(* CODESYS project mobject-core.library
   Author: mobject dev team
   Version: 0.10.0
   Title: mobject-core
   Placeholder: mobject-core
   DefaultNamespace: mobject-core
   Company: mobject

Project tree, tasks and I/O mapping:
  libraries: Tc2_Standard, * (Beckhoff Automation GmbH); Tc2_System, * (Beckhoff Automation GmbH); Tc2_Utilities, * (Beckhoff Automation GmbH); Tc3_JsonXml, * (Beckhoff Automation GmbH)
  mobject-collections/
    _Internal/
      Dictionary/
        Enumerator/
          function block DictionaryForwardEnumerator [ST]: FB_init, FB_exit, HandleEvent, IsValid, Key, MoveNext, Reset, TryGet, TryGetTo
        Node/
          function block DictionaryTreeNode [ST]: FB_init, FB_exit, CopyBufferToDestination, CopySourceToBuffer, CreateBuffer, DestroyBuffer, DataSize, DeepCopy, Equals, Height, Key, Left, NodeBufferPointer, NodeBufferSize, Reinitialize, Right, TryGet, TryGetTo
      Events/
        Collection/
          function block CollectionChangedEvent [ST]
          function block CollectionDisposedEvent [ST]
          function block CollectionEvent [ST]: FB_init, Target
        KeyValueCollection/
          function block KeyValueCollectionChangedEvent [ST]
          function block KeyValueCollectionDisposedEvent [ST]
          function block KeyValueCollectionEvent [ST]: FB_init, Target
      LinkedList/
        Enumerator/
          function block LinkedListForwardEnumerator [ST]: FB_init, FB_exit, HandleEvent, IsValid, MoveNext, Reset, TryGet, TryGetTo
        Node/
          function block LinkedListNode [ST]: FB_init, FB_exit, CopyBufferToDestination, CopySourceToBuffer, CreateBuffer, DestroyBuffer, DataSize, Equals, Next, Previous, TryGet, TryGetTo
      OrderedDictionary/
        Enumerator/
          function block OrderedDictionaryForwardEnumerator [ST]: FB_init, FB_exit, HandleEvent, IsValid, Key, MoveNext, Reset, TryGet, TryGetTo
        Node/
          function block OrderedDictionaryTreeNode [ST]: FB_init, FB_exit, CopyBufferToDestination, CopySourceToBuffer, CreateBuffer, DestroyBuffer, DataSize, DeepCopy, Equals, Height, Key, Left, Next, NodeBufferPointer, NodeBufferSize, Previous, Reinitialize, Right, TryGet, TryGetTo
      PriorityQueue/
    Dictionary/
      function block Dictionary [ST]: FB_exit, Balance, EmitChangedEvent, EmitDisposedEvent, FindMinimum, GetBalanceFactor, GetHeight, LeftRotate, RecursiveAddKeysInOrderToCollection, RecursiveAddNodesInOrderToCollection, RecursiveClear, RecursiveCountNodes, RecursiveDelete, RecursiveFind, RecursiveInsert, RightRotate, UpdateHeight, AddOrUpdate, Clear, ContainsKey, Count, GetEnumerator, GetKeys, GetKeyValueEnumerator, IsEmpty, OffEvent, OnceEvent, OnEvent, Remove, TryAdd, TryGetValue, TryGetValueTo
    Interfaces/
      Collections/
        Events/
          interface I_CollectionChangedEvent: Target
          interface I_CollectionDisposedEvent: Target
        Nodes/
          interface I_CollectionNode: DataSize, Equals, TryGet, TryGetTo
          interface I_LinkedListNode: Next, Previous
          interface I_ListNode
        interface I_Collection: AddItem, Clear, Contains, Count, IsEmpty, TryCopyTo, TryCopyToLocation, TryRemoveItem
        interface I_LinkedList: AddAfter, AddBefore, AddFirst, AddLast, Find, FindLast, First, Last, Remove, RemoveFirst, RemoveLast
        interface I_List: Capacity, GetIndexOf, TrimExcess, TryGetByIndex, TryGetToByIndex, TryInsert, TryRemoveAt
        interface I_Queue: Enqueue, TryDequeue, TryPeek
        interface I_Stack: Push, TryPeek, TryPop
      KeyValueCollections/
        Events/
          interface I_KeyValueCollectionChangedEvent: Target
          interface I_KeyValueCollectionDisposedEvent: Target
        Nodes/
          interface I_DictionaryTreeNode: DeepCopy, Height, Key, Left, NodeBufferPointer, NodeBufferSize, Reinitialize, Right
          interface I_OrderedDictionaryTreeNode: DeepCopy, Height, Key, Left, Next, NodeBufferPointer, NodeBufferSize, Previous, Reinitialize, Right
        interface I_Dictionary: AddOrUpdate, Clear, ContainsKey, GetKeys, IsEmpty, Remove, TryAdd, TryGetValue, TryGetValueTo
        interface I_KeyValueCollection
    LinkedList/
      function block LinkedList [ST]: FB_exit, AddNodeAfter, AddNodeBefore, AddNodeFirst, AddNodeLast, ContainsLinkedListNode, CreateNode, EmitChangedEvent, EmitDisposedEvent, FindFirstNodeWithValue, FindLastNodeWithValue, RemoveAllNodes, RemoveNode, AddAfter, AddBefore, AddFirst, AddItem, AddLast, Clear, Contains, Count, Find, FindLast, First, GetEnumerator, IsEmpty, Last, OffEvent, OnceEvent, OnEvent, Remove, RemoveFirst, RemoveLast, TryCopyTo, TryCopyToLocation, TryRemoveItem
    OrderedDictionary/
      function block OrderedDictionary [ST]: FB_exit, AddKeysInOrderToCollection, AddNodesInOrderToCollection, AddNodeToEnd, Balance, EmitChangedEvent, EmitDisposedEvent, FindMinimum, GetBalanceFactor, GetHeight, LeftRotate, RecursiveCountNodes, RecursiveDelete, RecursiveFind, RecursiveInsert, RemoveNodeFromLinkedList, ReplaceNodeInLinkedList, RightRotate, UpdateHeight, AddOrUpdate, Clear, ContainsKey, Count, GetEnumerator, GetKeys, GetKeyValueEnumerator, IsEmpty, OffEvent, OnceEvent, OnEvent, Remove, TryAdd, TryGetValue, TryGetValueTo
    Queue/
      function block Queue [ST]: FB_exit, EmitChangedEvent, EmitDisposedEvent, AddItem, Clear, Contains, Count, Enqueue, GetEnumerator, IsEmpty, OffEvent, OnceEvent, OnEvent, TryCopyTo, TryCopyToLocation, TryDequeue, TryPeek, TryRemoveItem
    Stack/
      function block Stack [ST]: FB_exit, EmitChangedEvent, EmitDisposedEvent, AddItem, Clear, Contains, Count, GetEnumerator, IsEmpty, OffEvent, OnceEvent, OnEvent, Push, TryCopyTo, TryCopyToLocation, TryPeek, TryPop, TryRemoveItem
  mobject-commands/
    _Internal/
      AsyncCommandStateMachine/
        function block AsyncCommandStateMachine [ST]: StateComplete_Aborting, StateComplete_Completing, StateComplete_Executing, StateComplete_Initializing, Abort, Error, ErrorId, Execute, IsAborted, IsAborting, IsCompleted, IsCompleting, IsErrored, IsExecuting, IsIdle, IsInitializing, Next
        interface I_AsyncCommandStateControl: Error, Next
    AsyncCommand/
      Interface/
        interface I_AsyncCommand: Abort, Busy, CyclicCall, Done, Error, ErrorId
      Runners/
        function block SingleAsyncCommandRunner [ST]: Busy, CyclicCall, Done, Error, ErrorId, ExecuteCommand
      function block AsyncCommand [ST]: OnAborted, OnAborting, OnCompleted, OnCompleting, OnErrored, OnExecuting, OnIdle, OnInitializing, Abort, Busy, CyclicCall, Done, Error, ErrorId, Execute
    Command/
      Interface/
        interface I_Command: Execute
  mobject-constants/
    global variables DatatypeLimits
  mobject-converters/
    Converters/
      BOOL_TO_/
        function TryConvert_BOOL_TO_BOOL [ST]
        function TryConvert_BOOL_TO_BYTE [ST]
        function TryConvert_BOOL_TO_DATE [ST]
        function TryConvert_BOOL_TO_Destination [ST]
        function TryConvert_BOOL_TO_DINT [ST]
        function TryConvert_BOOL_TO_DT [ST]
        function TryConvert_BOOL_TO_DWORD [ST]
        function TryConvert_BOOL_TO_INT [ST]
        function TryConvert_BOOL_TO_LINT [ST]
        function TryConvert_BOOL_TO_LREAL [ST]
        function TryConvert_BOOL_TO_LWORD [ST]
        function TryConvert_BOOL_TO_REAL [ST]
        function TryConvert_BOOL_TO_SINT [ST]
        function TryConvert_BOOL_TO_STRING [ST]
        function TryConvert_BOOL_TO_TIME [ST]
        function TryConvert_BOOL_TO_TOD [ST]
        function TryConvert_BOOL_TO_UDINT [ST]
        function TryConvert_BOOL_TO_UINT [ST]
        function TryConvert_BOOL_TO_ULINT [ST]
        function TryConvert_BOOL_TO_USINT [ST]
        function TryConvert_BOOL_TO_WORD [ST]
      BYTE_TO_/
        function TryConvert_BYTE_TO_BOOL [ST]
        function TryConvert_BYTE_TO_BYTE [ST]
        function TryConvert_BYTE_TO_DATE [ST]
        function TryConvert_BYTE_TO_Destination [ST]
        function TryConvert_BYTE_TO_DINT [ST]
        function TryConvert_BYTE_TO_DT [ST]
        function TryConvert_BYTE_TO_DWORD [ST]
        function TryConvert_BYTE_TO_INT [ST]
        function TryConvert_BYTE_TO_LINT [ST]
        function TryConvert_BYTE_TO_LREAL [ST]
        function TryConvert_BYTE_TO_LWORD [ST]
        function TryConvert_BYTE_TO_REAL [ST]
        function TryConvert_BYTE_TO_SINT [ST]
        function TryConvert_BYTE_TO_STRING [ST]
        function TryConvert_BYTE_TO_TIME [ST]
        function TryConvert_BYTE_TO_TOD [ST]
        function TryConvert_BYTE_TO_UDINT [ST]
        function TryConvert_BYTE_TO_UINT [ST]
        function TryConvert_BYTE_TO_ULINT [ST]
        function TryConvert_BYTE_TO_USINT [ST]
        function TryConvert_BYTE_TO_WORD [ST]
      DATE_TO_/
        function TryConvert_DATE_TO_BOOL [ST]
        function TryConvert_DATE_TO_BYTE [ST]
        function TryConvert_DATE_TO_DATE [ST]
        function TryConvert_DATE_TO_Destination [ST]
        function TryConvert_DATE_TO_DINT [ST]
        function TryConvert_DATE_TO_DT [ST]
        function TryConvert_DATE_TO_DWORD [ST]
        function TryConvert_DATE_TO_INT [ST]
        function TryConvert_DATE_TO_LINT [ST]
        function TryConvert_DATE_TO_LREAL [ST]
        function TryConvert_DATE_TO_LWORD [ST]
        function TryConvert_DATE_TO_REAL [ST]
        function TryConvert_DATE_TO_SINT [ST]
        function TryConvert_DATE_TO_STRING [ST]
        function TryConvert_DATE_TO_TIME [ST]
        function TryConvert_DATE_TO_TOD [ST]
        function TryConvert_DATE_TO_UDINT [ST]
        function TryConvert_DATE_TO_UINT [ST]
        function TryConvert_DATE_TO_ULINT [ST]
        function TryConvert_DATE_TO_USINT [ST]
        function TryConvert_DATE_TO_WORD [ST]
      DINT_TO_/
        function TryConvert_DINT_TO_BOOL [ST]
        function TryConvert_DINT_TO_BYTE [ST]
        function TryConvert_DINT_TO_DATE [ST]
        function TryConvert_DINT_TO_Destination [ST]
        function TryConvert_DINT_TO_DINT [ST]
        function TryConvert_DINT_TO_DT [ST]
        function TryConvert_DINT_TO_DWORD [ST]
        function TryConvert_DINT_TO_INT [ST]
        function TryConvert_DINT_TO_LINT [ST]
        function TryConvert_DINT_TO_LREAL [ST]
        function TryConvert_DINT_TO_LWORD [ST]
        function TryConvert_DINT_TO_REAL [ST]
        function TryConvert_DINT_TO_SINT [ST]
        function TryConvert_DINT_TO_STRING [ST]
        function TryConvert_DINT_TO_TIME [ST]
        function TryConvert_DINT_TO_TOD [ST]
        function TryConvert_DINT_TO_UDINT [ST]
        function TryConvert_DINT_TO_UINT [ST]
        function TryConvert_DINT_TO_ULINT [ST]
        function TryConvert_DINT_TO_USINT [ST]
        function TryConvert_DINT_TO_WORD [ST]
      DT_TO_/
        function TryConvert_DT_TO_BOOL [ST]
        function TryConvert_DT_TO_BYTE [ST]
        function TryConvert_DT_TO_DATE [ST]
        function TryConvert_DT_TO_Destination [ST]
        function TryConvert_DT_TO_DINT [ST]
        function TryConvert_DT_TO_DT [ST]
        function TryConvert_DT_TO_DWORD [ST]
        function TryConvert_DT_TO_INT [ST]
        function TryConvert_DT_TO_LINT [ST]
        function TryConvert_DT_TO_LREAL [ST]
        function TryConvert_DT_TO_LWORD [ST]
        function TryConvert_DT_TO_REAL [ST]
        function TryConvert_DT_TO_SINT [ST]
        function TryConvert_DT_TO_STRING [ST]
        function TryConvert_DT_TO_TIME [ST]
        function TryConvert_DT_TO_TOD [ST]
        function TryConvert_DT_TO_UDINT [ST]
        function TryConvert_DT_TO_UINT [ST]
        function TryConvert_DT_TO_ULINT [ST]
        function TryConvert_DT_TO_USINT [ST]
        function TryConvert_DT_TO_WORD [ST]
      DWORD_TO_/
        function TryConvert_DWORD_TO_BOOL [ST]
        function TryConvert_DWORD_TO_BYTE [ST]
        function TryConvert_DWORD_TO_DATE [ST]
        function TryConvert_DWORD_TO_Destination [ST]
        function TryConvert_DWORD_TO_DINT [ST]
        function TryConvert_DWORD_TO_DT [ST]
        function TryConvert_DWORD_TO_DWORD [ST]
        function TryConvert_DWORD_TO_INT [ST]
        function TryConvert_DWORD_TO_LINT [ST]
        function TryConvert_DWORD_TO_LREAL [ST]
        function TryConvert_DWORD_TO_LWORD [ST]
        function TryConvert_DWORD_TO_REAL [ST]
        function TryConvert_DWORD_TO_SINT [ST]
        function TryConvert_DWORD_TO_STRING [ST]
        function TryConvert_DWORD_TO_TIME [ST]
        function TryConvert_DWORD_TO_TOD [ST]
        function TryConvert_DWORD_TO_UDINT [ST]
        function TryConvert_DWORD_TO_UINT [ST]
        function TryConvert_DWORD_TO_ULINT [ST]
        function TryConvert_DWORD_TO_USINT [ST]
        function TryConvert_DWORD_TO_WORD [ST]
      INT_TO_/
        function TryConvert_INT_TO_BOOL [ST]
        function TryConvert_INT_TO_BYTE [ST]
        function TryConvert_INT_TO_DATE [ST]
        function TryConvert_INT_TO_Destination [ST]
        function TryConvert_INT_TO_DINT [ST]
        function TryConvert_INT_TO_DT [ST]
        function TryConvert_INT_TO_DWORD [ST]
        function TryConvert_INT_TO_INT [ST]
        function TryConvert_INT_TO_LINT [ST]
        function TryConvert_INT_TO_LREAL [ST]
        function TryConvert_INT_TO_LWORD [ST]
        function TryConvert_INT_TO_REAL [ST]
        function TryConvert_INT_TO_SINT [ST]
        function TryConvert_INT_TO_STRING [ST]
        function TryConvert_INT_TO_TIME [ST]
        function TryConvert_INT_TO_TOD [ST]
        function TryConvert_INT_TO_UDINT [ST]
        function TryConvert_INT_TO_UINT [ST]
        function TryConvert_INT_TO_ULINT [ST]
        function TryConvert_INT_TO_USINT [ST]
        function TryConvert_INT_TO_WORD [ST]
      LINT_TO_/
        function TryConvert_LINT_TO_BOOL [ST]
        function TryConvert_LINT_TO_BYTE [ST]
        function TryConvert_LINT_TO_DATE [ST]
        function TryConvert_LINT_TO_Destination [ST]
        function TryConvert_LINT_TO_DINT [ST]
        function TryConvert_LINT_TO_DT [ST]
        function TryConvert_LINT_TO_DWORD [ST]
        function TryConvert_LINT_TO_INT [ST]
        function TryConvert_LINT_TO_LINT [ST]
        function TryConvert_LINT_TO_LREAL [ST]
        function TryConvert_LINT_TO_LWORD [ST]
        function TryConvert_LINT_TO_REAL [ST]
        function TryConvert_LINT_TO_SINT [ST]
        function TryConvert_LINT_TO_STRING [ST]
        function TryConvert_LINT_TO_TIME [ST]
        function TryConvert_LINT_TO_TOD [ST]
        function TryConvert_LINT_TO_UDINT [ST]
        function TryConvert_LINT_TO_UINT [ST]
        function TryConvert_LINT_TO_ULINT [ST]
        function TryConvert_LINT_TO_USINT [ST]
        function TryConvert_LINT_TO_WORD [ST]
      LREAL_TO_/
        function TryConvert_LREAL_TO_BOOL [ST]
        function TryConvert_LREAL_TO_BYTE [ST]
        function TryConvert_LREAL_TO_DATE [ST]
        function TryConvert_LREAL_TO_Destination [ST]
        function TryConvert_LREAL_TO_DINT [ST]
        function TryConvert_LREAL_TO_DT [ST]
        function TryConvert_LREAL_TO_DWORD [ST]
        function TryConvert_LREAL_TO_INT [ST]
        function TryConvert_LREAL_TO_LINT [ST]
        function TryConvert_LREAL_TO_LREAL [ST]
        function TryConvert_LREAL_TO_LWORD [ST]
        function TryConvert_LREAL_TO_REAL [ST]
        function TryConvert_LREAL_TO_SINT [ST]
        function TryConvert_LREAL_TO_STRING [ST]
        function TryConvert_LREAL_TO_TIME [ST]
        function TryConvert_LREAL_TO_TOD [ST]
        function TryConvert_LREAL_TO_UDINT [ST]
        function TryConvert_LREAL_TO_UINT [ST]
        function TryConvert_LREAL_TO_ULINT [ST]
        function TryConvert_LREAL_TO_USINT [ST]
        function TryConvert_LREAL_TO_WORD [ST]
      LWORD_TO_/
        function TryConvert_LWORD_TO_BOOL [ST]
        function TryConvert_LWORD_TO_BYTE [ST]
        function TryConvert_LWORD_TO_DATE [ST]
        function TryConvert_LWORD_TO_Destination [ST]
        function TryConvert_LWORD_TO_DINT [ST]
        function TryConvert_LWORD_TO_DT [ST]
        function TryConvert_LWORD_TO_DWORD [ST]
        function TryConvert_LWORD_TO_INT [ST]
        function TryConvert_LWORD_TO_LINT [ST]
        function TryConvert_LWORD_TO_LREAL [ST]
        function TryConvert_LWORD_TO_LWORD [ST]
        function TryConvert_LWORD_TO_REAL [ST]
        function TryConvert_LWORD_TO_SINT [ST]
        function TryConvert_LWORD_TO_STRING [ST]
        function TryConvert_LWORD_TO_TIME [ST]
        function TryConvert_LWORD_TO_TOD [ST]
        function TryConvert_LWORD_TO_UDINT [ST]
        function TryConvert_LWORD_TO_UINT [ST]
        function TryConvert_LWORD_TO_ULINT [ST]
        function TryConvert_LWORD_TO_USINT [ST]
        function TryConvert_LWORD_TO_WORD [ST]
      REAL_TO_/
        function TryConvert_REAL_TO_BOOL [ST]
        function TryConvert_REAL_TO_BYTE [ST]
        function TryConvert_REAL_TO_DATE [ST]
        function TryConvert_REAL_TO_Destination [ST]
        function TryConvert_REAL_TO_DINT [ST]
        function TryConvert_REAL_TO_DT [ST]
        function TryConvert_REAL_TO_DWORD [ST]
        function TryConvert_REAL_TO_INT [ST]
        function TryConvert_REAL_TO_LINT [ST]
        function TryConvert_REAL_TO_LREAL [ST]
        function TryConvert_REAL_TO_LWORD [ST]
        function TryConvert_REAL_TO_REAL [ST]
        function TryConvert_REAL_TO_SINT [ST]
        function TryConvert_REAL_TO_STRING [ST]
        function TryConvert_REAL_TO_TIME [ST]
        function TryConvert_REAL_TO_TOD [ST]
        function TryConvert_REAL_TO_UDINT [ST]
        function TryConvert_REAL_TO_UINT [ST]
        function TryConvert_REAL_TO_ULINT [ST]
        function TryConvert_REAL_TO_USINT [ST]
        function TryConvert_REAL_TO_WORD [ST]
      SINT_TO_/
        function TryConvert_SINT_TO_BOOL [ST]
        function TryConvert_SINT_TO_BYTE [ST]
        function TryConvert_SINT_TO_DATE [ST]
        function TryConvert_SINT_TO_Destination [ST]
        function TryConvert_SINT_TO_DINT [ST]
        function TryConvert_SINT_TO_DT [ST]
        function TryConvert_SINT_TO_DWORD [ST]
        function TryConvert_SINT_TO_INT [ST]
        function TryConvert_SINT_TO_LINT [ST]
        function TryConvert_SINT_TO_LREAL [ST]
        function TryConvert_SINT_TO_LWORD [ST]
        function TryConvert_SINT_TO_REAL [ST]
        function TryConvert_SINT_TO_SINT [ST]
        function TryConvert_SINT_TO_STRING [ST]
        function TryConvert_SINT_TO_TIME [ST]
        function TryConvert_SINT_TO_TOD [ST]
        function TryConvert_SINT_TO_UDINT [ST]
        function TryConvert_SINT_TO_UINT [ST]
        function TryConvert_SINT_TO_ULINT [ST]
        function TryConvert_SINT_TO_USINT [ST]
        function TryConvert_SINT_TO_WORD [ST]
      STRING_TO_/
        function TryConvert_STRING_TO_BOOL [ST]
        function TryConvert_STRING_TO_BYTE [ST]
        function TryConvert_STRING_TO_DATE [ST]
        function TryConvert_STRING_TO_Destination [ST]
        function TryConvert_STRING_TO_DINT [ST]
        function TryConvert_STRING_TO_DT [ST]
        function TryConvert_STRING_TO_DWORD [ST]
        function TryConvert_STRING_TO_INT [ST]
        function TryConvert_STRING_TO_LINT [ST]
        function TryConvert_STRING_TO_LREAL [ST]
        function TryConvert_STRING_TO_LWORD [ST]
        function TryConvert_STRING_TO_REAL [ST]
        function TryConvert_STRING_TO_SINT [ST]
        function TryConvert_STRING_TO_STRING [ST]
        function TryConvert_STRING_TO_TIME [ST]
        function TryConvert_STRING_TO_TOD [ST]
        function TryConvert_STRING_TO_UDINT [ST]
        function TryConvert_STRING_TO_UINT [ST]
        function TryConvert_STRING_TO_ULINT [ST]
        function TryConvert_STRING_TO_USINT [ST]
        function TryConvert_STRING_TO_WORD [ST]
      TIME_TO_/
        function TryConvert_TIME_TO_BOOL [ST]
        function TryConvert_TIME_TO_BYTE [ST]
        function TryConvert_TIME_TO_DATE [ST]
        function TryConvert_TIME_TO_Destination [ST]
        function TryConvert_TIME_TO_DINT [ST]
        function TryConvert_TIME_TO_DT [ST]
        function TryConvert_TIME_TO_DWORD [ST]
        function TryConvert_TIME_TO_INT [ST]
        function TryConvert_TIME_TO_LINT [ST]
        function TryConvert_TIME_TO_LREAL [ST]
        function TryConvert_TIME_TO_LWORD [ST]
        function TryConvert_TIME_TO_REAL [ST]
        function TryConvert_TIME_TO_SINT [ST]
        function TryConvert_TIME_TO_STRING [ST]
        function TryConvert_TIME_TO_TIME [ST]
        function TryConvert_TIME_TO_TOD [ST]
        function TryConvert_TIME_TO_UDINT [ST]
        function TryConvert_TIME_TO_UINT [ST]
        function TryConvert_TIME_TO_ULINT [ST]
        function TryConvert_TIME_TO_USINT [ST]
        function TryConvert_TIME_TO_WORD [ST]
      TOD_TO_/
        function TryConvert_TOD_TO_BOOL [ST]
        function TryConvert_TOD_TO_BYTE [ST]
        function TryConvert_TOD_TO_DATE [ST]
        function TryConvert_TOD_TO_Destination [ST]
        function TryConvert_TOD_TO_DINT [ST]
        function TryConvert_TOD_TO_DT [ST]
        function TryConvert_TOD_TO_DWORD [ST]
        function TryConvert_TOD_TO_INT [ST]
        function TryConvert_TOD_TO_LINT [ST]
        function TryConvert_TOD_TO_LREAL [ST]
        function TryConvert_TOD_TO_LWORD [ST]
        function TryConvert_TOD_TO_REAL [ST]
        function TryConvert_TOD_TO_SINT [ST]
        function TryConvert_TOD_TO_STRING [ST]
        function TryConvert_TOD_TO_TIME [ST]
        function TryConvert_TOD_TO_TOD [ST]
        function TryConvert_TOD_TO_UDINT [ST]
        function TryConvert_TOD_TO_UINT [ST]
        function TryConvert_TOD_TO_ULINT [ST]
        function TryConvert_TOD_TO_USINT [ST]
        function TryConvert_TOD_TO_WORD [ST]
      UDINT_TO_/
        function TryConvert_UDINT_TO_BOOL [ST]
        function TryConvert_UDINT_TO_BYTE [ST]
        function TryConvert_UDINT_TO_DATE [ST]
        function TryConvert_UDINT_TO_Destination [ST]
        function TryConvert_UDINT_TO_DINT [ST]
        function TryConvert_UDINT_TO_DT [ST]
        function TryConvert_UDINT_TO_DWORD [ST]
        function TryConvert_UDINT_TO_INT [ST]
        function TryConvert_UDINT_TO_LINT [ST]
        function TryConvert_UDINT_TO_LREAL [ST]
        function TryConvert_UDINT_TO_LWORD [ST]
        function TryConvert_UDINT_TO_REAL [ST]
        function TryConvert_UDINT_TO_SINT [ST]
        function TryConvert_UDINT_TO_STRING [ST]
        function TryConvert_UDINT_TO_TIME [ST]
        function TryConvert_UDINT_TO_TOD [ST]
        function TryConvert_UDINT_TO_UDINT [ST]
        function TryConvert_UDINT_TO_UINT [ST]
        function TryConvert_UDINT_TO_ULINT [ST]
        function TryConvert_UDINT_TO_USINT [ST]
        function TryConvert_UDINT_TO_WORD [ST]
      UINT_TO_/
        function TryConvert_UINT_TO_BOOL [ST]
        function TryConvert_UINT_TO_BYTE [ST]
        function TryConvert_UINT_TO_DATE [ST]
        function TryConvert_UINT_TO_Destination [ST]
        function TryConvert_UINT_TO_DINT [ST]
        function TryConvert_UINT_TO_DT [ST]
        function TryConvert_UINT_TO_DWORD [ST]
        function TryConvert_UINT_TO_INT [ST]
        function TryConvert_UINT_TO_LINT [ST]
        function TryConvert_UINT_TO_LREAL [ST]
        function TryConvert_UINT_TO_LWORD [ST]
        function TryConvert_UINT_TO_REAL [ST]
        function TryConvert_UINT_TO_SINT [ST]
        function TryConvert_UINT_TO_STRING [ST]
        function TryConvert_UINT_TO_TIME [ST]
        function TryConvert_UINT_TO_TOD [ST]
        function TryConvert_UINT_TO_UDINT [ST]
        function TryConvert_UINT_TO_UINT [ST]
        function TryConvert_UINT_TO_ULINT [ST]
        function TryConvert_UINT_TO_USINT [ST]
        function TryConvert_UINT_TO_WORD [ST]
      ULINT_TO_/
        function TryConvert_ULINT_TO_BOOL [ST]
        function TryConvert_ULINT_TO_BYTE [ST]
        function TryConvert_ULINT_TO_DATE [ST]
        function TryConvert_ULINT_TO_Destination [ST]
        function TryConvert_ULINT_TO_DINT [ST]
        function TryConvert_ULINT_TO_DT [ST]
        function TryConvert_ULINT_TO_DWORD [ST]
        function TryConvert_ULINT_TO_INT [ST]
        function TryConvert_ULINT_TO_LINT [ST]
        function TryConvert_ULINT_TO_LREAL [ST]
        function TryConvert_ULINT_TO_LWORD [ST]
        function TryConvert_ULINT_TO_REAL [ST]
        function TryConvert_ULINT_TO_SINT [ST]
        function TryConvert_ULINT_TO_STRING [ST]
        function TryConvert_ULINT_TO_TIME [ST]
        function TryConvert_ULINT_TO_TOD [ST]
        function TryConvert_ULINT_TO_UDINT [ST]
        function TryConvert_ULINT_TO_UINT [ST]
        function TryConvert_ULINT_TO_ULINT [ST]
        function TryConvert_ULINT_TO_USINT [ST]
        function TryConvert_ULINT_TO_WORD [ST]
      USINT_TO_/
        function TryConvert_USINT_TO_BOOL [ST]
        function TryConvert_USINT_TO_BYTE [ST]
        function TryConvert_USINT_TO_DATE [ST]
        function TryConvert_USINT_TO_Destination [ST]
        function TryConvert_USINT_TO_DINT [ST]
        function TryConvert_USINT_TO_DT [ST]
        function TryConvert_USINT_TO_DWORD [ST]
        function TryConvert_USINT_TO_INT [ST]
        function TryConvert_USINT_TO_LINT [ST]
        function TryConvert_USINT_TO_LREAL [ST]
        function TryConvert_USINT_TO_LWORD [ST]
        function TryConvert_USINT_TO_REAL [ST]
        function TryConvert_USINT_TO_SINT [ST]
        function TryConvert_USINT_TO_STRING [ST]
        function TryConvert_USINT_TO_TIME [ST]
        function TryConvert_USINT_TO_TOD [ST]
        function TryConvert_USINT_TO_UDINT [ST]
        function TryConvert_USINT_TO_UINT [ST]
        function TryConvert_USINT_TO_ULINT [ST]
        function TryConvert_USINT_TO_USINT [ST]
        function TryConvert_USINT_TO_WORD [ST]
      WORD_TO_/
        function TryConvert_WORD_TO_BOOL [ST]
        function TryConvert_WORD_TO_BYTE [ST]
        function TryConvert_WORD_TO_DATE [ST]
        function TryConvert_WORD_TO_Destination [ST]
        function TryConvert_WORD_TO_DINT [ST]
        function TryConvert_WORD_TO_DT [ST]
        function TryConvert_WORD_TO_DWORD [ST]
        function TryConvert_WORD_TO_INT [ST]
        function TryConvert_WORD_TO_LINT [ST]
        function TryConvert_WORD_TO_LREAL [ST]
        function TryConvert_WORD_TO_LWORD [ST]
        function TryConvert_WORD_TO_REAL [ST]
        function TryConvert_WORD_TO_SINT [ST]
        function TryConvert_WORD_TO_STRING [ST]
        function TryConvert_WORD_TO_TIME [ST]
        function TryConvert_WORD_TO_TOD [ST]
        function TryConvert_WORD_TO_UDINT [ST]
        function TryConvert_WORD_TO_UINT [ST]
        function TryConvert_WORD_TO_ULINT [ST]
        function TryConvert_WORD_TO_USINT [ST]
        function TryConvert_WORD_TO_WORD [ST]
      function TryConvert_Source_TO_Destination [ST]
  mobject-datatypes/
    _Internal/
      Datatype/
        Interface/
          interface I_AliasDatatype: BaseDatatype
          interface I_ArrayDatatype: Dimention, TryGetLowerBound, TryGetUpperBound, TryResolveAs1DArrayDatatype, TryResolveAs2DArrayDatatype, TryResolveAs3DArrayDatatype
          interface I_ArrayDatatype_1D: TryGetElementAsDatatypeByIndex
          interface I_ArrayDatatype_2D: TryGetElementAsDatatypeByIndex
          interface I_ArrayDatatype_3D: TryGetElementAsDatatypeByIndex
          interface I_Datatype: Accept, Address, ClearReference, Clone, IsEquivalentTo, IsNull, IsUserDefined, Root, SerializeTypeWith, Size, TryConvertTo, TryConvertTo_, TryCopyFrom, TryDeserializeFrom, TryMakeReferenceTo, TryResolveAs_ANY, TryResolveAs_BIT, TryResolveAs_BOOL, TryResolveAs_BYTE, TryResolveAs_DINT, TryResolveAs_DT, TryResolveAs_DWORD, TryResolveAs_INT, TryResolveAs_LINT, TryResolveAs_LREAL, TryResolveAs_LWORD, TryResolveAs_PVOID, TryResolveAs_REAL, TryResolveAs_REFERENCE_TO, TryResolveAs_SINT, TryResolveAs_STRING, TryResolveAs_TIME_OF_DAY, TryResolveAs_TOD, TryResolveAs_UDINT, TryResolveAs_UINT, TryResolveAs_ULINT, TryResolveAs_USINT, TryResolveAs_WORD, TryResolveAsAliasDatatype, TryResolveAsArrayDatatype, TryResolveAsBitDatatype, TryResolveAsEnumDatatype, TryResolveAsInterfaceDatatype, TryResolveAsStructuredDatatype, TryResolveAsUserDefinedDatatype, TypeName
          interface I_EnumDatatype
          interface I_InterfaceDatatype: Identifier, TryCopyContentFrom
          interface I_NumericDatatype: IsFloat, IsSigned
          interface I_StructuredDatatype
          interface I_UserDefinedDatatype: Identifier
        function block AliasDatatypeBase [ST]: AddBaseDatatype, OnSerializeTypeWith, BaseDatatype, IsEquivalentTo, Root, SerializeWith, TryConvertTo, TryConvertTo_, TryDeserializeFrom, TryResolveAsAliasDatatype, TypeName
        function block ArrayDatatypeBase_1D [ST]: SerializeBaseType, OnSerializeArrayValues, OnSerializeTypeWith, TryDeserializeArrayValues, BaseDatatype, Dimention, Identifier, Length, SerializeWith, TryDeserializeFrom, TryGetElementAsDatatypeByIndex, TryGetLowerBound, TryGetUpperBound, TryResolveAs1DArrayDatatype, TryResolveAs2DArrayDatatype, TryResolveAs3DArrayDatatype, TryResolveAsArrayDatatype, TypeName
        function block ArrayDatatypeBase_2D [ST]: SerializeBaseType, OnSerializeArrayValues, OnSerializeTypeWith, TryDeserializeArrayValues, BaseDatatype, Dimention, Identifier, Length, SerializeWith, TryDeserializeFrom, TryGetElementAsDatatypeByIndex, TryGetLowerBound, TryGetUpperBound, TryResolveAs1DArrayDatatype, TryResolveAs2DArrayDatatype, TryResolveAs3DArrayDatatype, TryResolveAsArrayDatatype, TypeName
        function block ArrayDatatypeBase_3D [ST]: SerializeBaseType, OnSerializeArrayValues, OnSerializeTypeWith, TryDeserializeArrayValues, BaseDatatype, Dimention, Identifier, Length, SerializeWith, TryDeserializeFrom, TryGetElementAsDatatypeByIndex, TryGetLowerBound, TryGetUpperBound, TryResolveAs1DArrayDatatype, TryResolveAs2DArrayDatatype, TryResolveAs3DArrayDatatype, TryResolveAsArrayDatatype, TypeName
        function block DatatypeBase [ST]: OnSerializeTypeWith, Accept, Address, ClearReference, Clone, IsEquivalentTo, IsNull, IsUserDefined, Root, SerializeTypeWith, SerializeWith, Size, TryConvertTo, TryConvertTo_, TryCopyFrom, TryDeserializeFrom, TryMakeReferenceTo, TryResolveAs_ANY, TryResolveAs_BIT, TryResolveAs_BOOL, TryResolveAs_BYTE, TryResolveAs_DINT, TryResolveAs_DT, TryResolveAs_DWORD, TryResolveAs_INT, TryResolveAs_LINT, TryResolveAs_LREAL, TryResolveAs_LWORD, TryResolveAs_PVOID, TryResolveAs_REAL, TryResolveAs_REFERENCE_TO, TryResolveAs_SINT, TryResolveAs_STRING, TryResolveAs_TIME_OF_DAY, TryResolveAs_TOD, TryResolveAs_UDINT, TryResolveAs_UINT, TryResolveAs_ULINT, TryResolveAs_USINT, TryResolveAs_WORD, TryResolveAsAliasDatatype, TryResolveAsArrayDatatype, TryResolveAsBitDatatype, TryResolveAsEnumDatatype, TryResolveAsInterfaceDatatype, TryResolveAsStructuredDatatype, TryResolveAsUserDefinedDatatype, TypeName
        function block EnumDatatypeBase [ST]: CreateEnumError, SerializeBaseType, SerializeEnums, AddBaseDatatype, AddEnumeration, IsEnumeratorValueEqual, OnSerializeTypeWith, BaseDatatype, IsEquivalentTo, Root, SerializeWith, TryDeserializeFrom, TryResolveAsEnumDatatype, TypeName
        function block InterfaceDatatypeBase [ST]: OnSerializeTypeWith, Identifier, IsUserDefined, TryCopyContentFrom, TryCopyFrom, TryResolveAsInterfaceDatatype, TypeName
        function block NumericDatatypeBase [ST]: OnSerializeTypeWith, SerializeMaxValue, SerializeMinValue, IsEven, IsFloat, IsOdd, IsSigned
        function block StructuredDatatypeBase [ST]: AddMember, OnSerializeTypeWith, Accept, Members, SerializeWith, TryDeserializeFrom, TryResolveAsStructuredDatatype, TypeName
        function block UserDefinedDatatypeBase [ST]: OnSerializeTypeWith, Identifier, IsEquivalentTo, IsUserDefined, TryCopyFrom, TryResolveAsUserDefinedDatatype
      Errors/
        function block UnknownEnumerationError [ST]: FB_init, ErrorType, Message
      Events/
        function block AliasDatatypeAddedEvent [ST]: FB_init, Target
        function block ArrayDatatypeAddedEvent [ST]: FB_init, Target
        function block DatatypeAddedEvent [ST]: FB_init, Target
        function block EnumDatatypeAddedEvent [ST]: FB_init, Target
        function block InterfaceDatatypeAddedEvent [ST]: FB_init, Target
        function block StructuredDatatypeAddedEvent [ST]: FB_init, Target
      StructureMembers/
        Host/
          function block StructureMemberHost [ST]: Accept, AddMember, GetMemberEnumerator, SerializeTypeWith, SerializeWith, TryDeserializeFrom, TryGetMemberByName
        Interface/
          interface I_HostStructureMembers: Members
          interface I_StructureMembers: Accept, GetMemberEnumerator, TryGetMemberByName
    DatatypeOperations/
      Collection/
        function block DatatypeOperations [ST]: FB_exit, CreateMemoryCopyOperation, CreateSafeMemoryCopyOperation, CreateWriteBitToBoolOperation, CreateWriteBoolToBitOperation, AddMemoryCopyOperation, AddSafeMemoryCopyOperation, AddWriteBitToBoolOperation, AddWriteBoolToBitOperation, Clear, Execute
      Interface/
        interface I_DatatypeOperation: Execute
      function block MemCopyOperation [ST]: FB_init, Execute
      function block SafeMemCopyOperation [ST]: FB_init, Execute
      function block WriteBitToBoolOperation [ST]: FB_init, Execute
      function block WriteBoolToBitOperation [ST]: FB_init, Execute
    Datatypes/
      Base/
        function block Datatypes [ST]: AcceptAlias, AcceptArrays, AcceptEnum, AcceptInterface, AcceptPrimative, AcceptStructures, SerializeAliasTypeWith, SerializeArrayTypeWith, SerializeEnumsTypeWith, SerializeInterfaceTypeWith, SerializePrimitiveTypeWith, SerializeStructuresTypeWith, EmitOnAliasDatatypeAddedEvent, EmitOnArrayDatatypeAddedEvent, EmitOnDatatypeAddedEvent, EmitOnEnumDatatypeAddedEvent, EmitOnInterfaceDatatypeAddedEvent, EmitOnStructuredDatatypeAddedEvent, Accept, OffEvent, OnceEvent, OnEvent, RegisterDatatype, SerializeTypeWith, TryGetAliasByIdentifier, TryGetArrayByIdentifier, TryGetEnumByIdentifier, TryGetInterfaceByIdentifier, TryGetPrimitiveByTypeName, TryGetStructureByIdentifier
      Events/
        interface I_AliasDatatypeAddedEvent: Target
        interface I_ArrayDatatypeAddedEvent: Target
        interface I_DatatypeAddedEvent: Target
        interface I_EnumDatatypeAddedEvent: Target
        interface I_InterfaceDatatypeAddedEvent: Target
        interface I_StructuredDatatypeAddedEvent: Target
      Interface/
        interface I_Datatypes: Accept, RegisterDatatype, SerializeTypeWith, TryGetAliasByIdentifier, TryGetArrayByIdentifier, TryGetEnumByIdentifier, TryGetInterfaceByIdentifier, TryGetPrimitiveByTypeName, TryGetStructureByIdentifier
    DatatypeVisitor/
      interface I_DatatypeVisitor: VisitDatatype
    Functions/
      function GetByteOffset [ST]
    Primitive/
      Interfaces/
        interface I_ANY: CanBecome, Clear, IsResolved, TryBecome
        interface I_BIT: BitOffset, ByteOffset, Parent, Value
        interface I_BOOL: Value
        interface I_BYTE: Value
        interface I_DINT: Value
        interface I_DT: Value
        interface I_DWORD: Value
        interface I_INT: Value
        interface I_LINT: Value
        interface I_LREAL: Value
        interface I_LWORD: Value
        interface I_PVOID: Value
        interface I_REAL: Value
        interface I_REFERENCE_TO: IsValidReference
        interface I_SINT: Value
        interface I_STRING: Value
        interface I_TIME_OF_DAY: Value
        interface I_TOD: Value
        interface I_UDINT: Value
        interface I_UINT: Value
        interface I_ULINT: Value
        interface I_USINT: Value
        interface I_WORD: Value
      function block _ANY [ST]: FB_exit, ClearResolvedDatatype, CreateResolvedDatatype, Accept, Address, CanBecome, Clear, ClearReference, Clone, IsEquivalentTo, IsNull, IsResolved, IsUserDefined, Root, SerializeTypeWith, SerializeWith, Size, TryBecome, TryConvertTo, TryConvertTo_, TryCopyFrom, TryDeserializeFrom, TryMakeReferenceTo, TryResolveAs_ANY, TryResolveAs_BIT, TryResolveAs_BOOL, TryResolveAs_BYTE, TryResolveAs_DINT, TryResolveAs_DT, TryResolveAs_DWORD, TryResolveAs_INT, TryResolveAs_LINT, TryResolveAs_LREAL, TryResolveAs_LWORD, TryResolveAs_PVOID, TryResolveAs_REAL, TryResolveAs_REFERENCE_TO, TryResolveAs_SINT, TryResolveAs_STRING, TryResolveAs_TIME_OF_DAY, TryResolveAs_TOD, TryResolveAs_UDINT, TryResolveAs_UINT, TryResolveAs_ULINT, TryResolveAs_USINT, TryResolveAs_WORD, TryResolveAsAliasDatatype, TryResolveAsArrayDatatype, TryResolveAsBitDatatype, TryResolveAsEnumDatatype, TryResolveAsInterfaceDatatype, TryResolveAsStructuredDatatype, TryResolveAsUserDefinedDatatype, TypeName
      function block _BIT [ST]: GetBitValue, SetBitValue, Address, BitOffset, ByteOffset, ClearReference, Clone, MakeReferenceTo, Parent, SerializeWith, Size, TryConvertTo, TryConvertTo_, TryDeserializeFrom, TryMakeReferenceTo, TryResolveAs_BIT, TypeName, Value
      function block _BOOL [ST]: FB_init, Address, ClearReference, Clone, MakeReferenceTo, SerializeWith, Size, TryConvertTo, TryConvertTo_, TryDeserializeFrom, TryMakeReferenceTo, TryResolveAs_BOOL, TypeName, Value
      function block _BYTE [ST]: FB_init, SerializeMaxValue, SerializeMinValue, Address, ClearReference, Clone, IsEven, IsFloat, IsSigned, MakeReferenceTo, MaxValue, MinValue, SerializeWith, Size, TryConvertTo, TryConvertTo_, TryDeserializeFrom, TryMakeReferenceTo, TryResolveAs_BYTE, TypeName, Value
      function block _DINT [ST]: FB_init, SerializeMaxValue, SerializeMinValue, Address, ClearReference, Clone, IsEven, IsFloat, IsSigned, MakeReferenceTo, MaxValue, MinValue, SerializeWith, Size, TryConvertTo, TryConvertTo_, TryDeserializeFrom, TryMakeReferenceTo, TryResolveAs_DINT, TypeName, Value
      function block _DT [ST]: FB_init, Address, ClearReference, Clone, MakeReferenceTo, SerializeWith, Size, TryConvertTo, TryConvertTo_, TryDeserializeFrom, TryMakeReferenceTo, TryResolveAs_DT, TypeName, Value
      function block _DWORD [ST]: FB_init, SerializeMaxValue, SerializeMinValue, Address, ClearReference, Clone, IsEven, IsFloat, IsSigned, MakeReferenceTo, MaxValue, MinValue, SerializeWith, Size, TryConvertTo, TryConvertTo_, TryDeserializeFrom, TryMakeReferenceTo, TryResolveAs_DWORD, TypeName, Value
      function block _INT [ST]: FB_init, SerializeMaxValue, SerializeMinValue, Address, ClearReference, Clone, IsEven, IsFloat, IsSigned, MakeReferenceTo, MaxValue, MinValue, SerializeWith, Size, TryConvertTo, TryConvertTo_, TryDeserializeFrom, TryMakeReferenceTo, TryResolveAs_INT, TypeName, Value
      function block _LINT [ST]: FB_init, SerializeMaxValue, SerializeMinValue, Address, ClearReference, Clone, IsEven, IsFloat, IsSigned, MakeReferenceTo, MaxValue, MinValue, SerializeWith, Size, TryConvertTo, TryConvertTo_, TryDeserializeFrom, TryMakeReferenceTo, TryResolveAs_LINT, TypeName, Value
      function block _LREAL [ST]: FB_init, SerializeMaxValue, SerializeMinValue, Address, ClearReference, Clone, IsEven, IsFloat, IsOdd, IsSigned, MakeReferenceTo, MaxValue, MinValue, SerializeWith, Size, TryConvertTo, TryConvertTo_, TryDeserializeFrom, TryMakeReferenceTo, TryResolveAs_LREAL, TypeName, Value
      function block _LWORD [ST]: FB_init, SerializeMaxValue, SerializeMinValue, Address, ClearReference, Clone, IsEven, IsFloat, IsSigned, MakeReferenceTo, MaxValue, MinValue, SerializeWith, Size, TryConvertTo, TryConvertTo_, TryDeserializeFrom, TryMakeReferenceTo, TryResolveAs_LWORD, TypeName, Value
      function block _NULL [ST]: Address, ClearReference, Clone, IsNull, SerializeWith, Size, TryDeserializeFrom, TryMakeReferenceTo, TypeName
      function block _PVOID [ST]: Address, ClearReference, Clone, MakeReferenceTo, SerializeWith, Size, TryDeserializeFrom, TryMakeReferenceTo, TryResolveAs_PVOID, TypeName, Value
      function block _REAL [ST]: FB_init, SerializeMaxValue, SerializeMinValue, Address, ClearReference, Clone, IsEven, IsFloat, IsOdd, IsSigned, MakeReferenceTo, MaxValue, MinValue, SerializeWith, Size, TryConvertTo, TryConvertTo_, TryDeserializeFrom, TryMakeReferenceTo, TryResolveAs_REAL, TypeName, Value
      function block _REFERENCE_TO [ST]: FB_Init, Accept, Address, ClearReference, Clone, IsEquivalentTo, IsNull, IsUserDefined, IsValidReference, Root, SerializeTypeWith, SerializeWith, Size, TryConvertTo, TryConvertTo_, TryCopyFrom, TryDeserializeFrom, TryMakeReferenceTo, TryResolveAs_ANY, TryResolveAs_BIT, TryResolveAs_BOOL, TryResolveAs_BYTE, TryResolveAs_DINT, TryResolveAs_DT, TryResolveAs_DWORD, TryResolveAs_INT, TryResolveAs_LINT, TryResolveAs_LREAL, TryResolveAs_LWORD, TryResolveAs_PVOID, TryResolveAs_REAL, TryResolveAs_REFERENCE_TO, TryResolveAs_SINT, TryResolveAs_STRING, TryResolveAs_TIME_OF_DAY, TryResolveAs_TOD, TryResolveAs_UDINT, TryResolveAs_UINT, TryResolveAs_ULINT, TryResolveAs_USINT, TryResolveAs_WORD, TryResolveAsAliasDatatype, TryResolveAsArrayDatatype, TryResolveAsBitDatatype, TryResolveAsEnumDatatype, TryResolveAsInterfaceDatatype, TryResolveAsStructuredDatatype, TryResolveAsUserDefinedDatatype, TypeName
      function block _SINT [ST]: FB_init, SerializeMaxValue, SerializeMinValue, Address, ClearReference, Clone, IsEven, IsFloat, IsSigned, MakeReferenceTo, MaxValue, MinValue, SerializeWith, Size, TryConvertTo, TryConvertTo_, TryDeserializeFrom, TryMakeReferenceTo, TryResolveAs_SINT, TypeName, Value
      function block _STRING [ST]: FB_init, Address, ClearReference, Clone, Length, MakeReferenceTo, SerializeWith, Size, TryConvertTo, TryConvertTo_, TryDeserializeFrom, TryMakeReferenceTo, TryResolveAs_STRING, TypeName, Value
      function block _TIME_OF_DAY [ST]: FB_init, Address, ClearReference, Clone, MakeReferenceTo, SerializeWith, Size, TryDeserializeFrom, TryMakeReferenceTo, TryResolveAs_TIME_OF_DAY, TypeName, Value
      function block _TOD [ST]: FB_init, Address, ClearReference, Clone, MakeReferenceTo, SerializeWith, Size, TryConvertTo, TryConvertTo_, TryDeserializeFrom, TryMakeReferenceTo, TryResolveAs_TOD, TypeName, Value
      function block _UDINT [ST]: FB_init, SerializeMaxValue, SerializeMinValue, Address, ClearReference, Clone, IsEven, IsFloat, IsSigned, MakeReferenceTo, MaxValue, MinValue, SerializeWith, Size, TryConvertTo, TryConvertTo_, TryDeserializeFrom, TryMakeReferenceTo, TryResolveAs_UDINT, TypeName, Value
      function block _UINT [ST]: FB_init, SerializeMaxValue, SerializeMinValue, Address, ClearReference, Clone, IsEven, IsFloat, IsSigned, MakeReferenceTo, MaxValue, MinValue, SerializeWith, Size, TryConvertTo, TryConvertTo_, TryDeserializeFrom, TryMakeReferenceTo, TryResolveAs_UINT, TypeName, Value
      function block _ULINT [ST]: FB_init, SerializeMaxValue, SerializeMinValue, Address, ClearReference, Clone, IsEven, IsFloat, IsSigned, MakeReferenceTo, MaxValue, MinValue, SerializeWith, Size, TryConvertTo, TryConvertTo_, TryDeserializeFrom, TryMakeReferenceTo, TryResolveAs_ULINT, TypeName, Value
      function block _USINT [ST]: FB_init, SerializeMaxValue, SerializeMinValue, Address, ClearReference, Clone, IsEven, IsFloat, IsSigned, MakeReferenceTo, MaxValue, MinValue, SerializeWith, Size, TryConvertTo, TryConvertTo_, TryDeserializeFrom, TryMakeReferenceTo, TryResolveAs_USINT, TypeName, Value
      function block _WORD [ST]: FB_init, SerializeMaxValue, SerializeMinValue, Address, ClearReference, Clone, IsEven, IsFloat, IsSigned, MakeReferenceTo, MaxValue, MinValue, SerializeWith, Size, TryConvertTo, TryConvertTo_, TryDeserializeFrom, TryMakeReferenceTo, TryResolveAs_WORD, TypeName, Value
  mobject-deserialization/
    DeserializationFeedback/
      function block DeserializerFeedback [ST]: FB_exit, DisposeErrors, FirstError, HasError, LogDeserializationFailedError, LogError, LogIncorrectKeyTypeError, LogIncorrectTypeError, LogInvalidKeyError, LogMissingKeyError, Reset, SerializeWith
    Errors/
      CustomError/
        function block CustomDeserializationFailedError [ST]: FB_init, ErrorType, Message
      IncorrectType/
        function block IncorrectKeyTypeDeserializationError [ST]: FB_init, Message
        function block IncorrectTypeDeserializationError [ST]: FB_init, ErrorType, Message
      Invalid Index/
        function block InvalidArrayIndexDeserializationError [ST]: FB_init, ErrorType, Message
      Invalid Key/
        function block InvalidKeyDeserializationError [ST]: ErrorType, Message
      Missing Key/
        function block MissingKeyDeserializationError [ST]: FB_init, ErrorType, Message
      function block DeserializationErrorFactory [ST]: CreateCustomDeserializationFailedError, CreateIncorrectKeyTypeError, CreateIncorrectTypeError, CreateInvalidArrayIndexError, CreateInvalidKeyError, CreateMissingKeyError
    GarbageCollector/
      function block DeserializerGarbageCollector [ST]: FB_exit, DisposeAll, Deregister, Execute, Register
      interface I_DeserializerGarbageCollector: Deregister, Register
    Interfaces/
      interface I_Deserializable: TryDeserializeFrom
      interface I_Deserializer: Clone, GetArray, GetArrayEnumerator, GetElementByIndex, GetKeyArray, GetKeyObject, GetObject, GetObjectEnumerator, TryDeserializeKeyToObject, TryDeserializeToObject, TryGetBase64, TryGetBool, TryGetByte, TryGetDateTime, TryGetDcTime, TryGetDint, TryGetDword, TryGetElementByIndex, TryGetFileTime, TryGetHexAsBytes, TryGetInt, TryGetKeyBase64, TryGetKeyBool, TryGetKeyByte, TryGetKeyDateTime, TryGetKeyDcTime, TryGetKeyDint, TryGetKeyDword, TryGetKeyFileTime, TryGetKeyHexAsBytes, TryGetKeyInt, TryGetKeyLint, TryGetKeyLreal, TryGetKeyLtime, TryGetKeyLword, TryGetKeyReal, TryGetKeySint, TryGetKeyString, TryGetKeyStringEx, TryGetKeyTime, TryGetKeyTod, TryGetKeyUdint, TryGetKeyUint, TryGetKeyUlint, TryGetKeyUsint, TryGetKeyWord, TryGetLint, TryGetLreal, TryGetLtime, TryGetLword, TryGetReal, TryGetSint, TryGetString, TryGetStringEx, TryGetTime, TryGetTod, TryGetUdint, TryGetUint, TryGetUlint, TryGetUsint, TryGetWord
      interface I_DeserializerArrayForwardEnumerator: Current, Index, IsValid, MoveNext
      interface I_DeserializerFeedback: LogDeserializationFailedError, LogError, LogIncorrectKeyTypeError, LogIncorrectTypeError, LogInvalidKeyError, LogMissingKeyError
      interface I_DeserializerObjectForwardEnumerator: Current, IsValid, Key, MoveNext
  mobject-disposable/
    Disposable/
      function block Disposable [ST]: FB_exit, Dispose
    Interfaces/
      interface I_Disposable: Dispose
  mobject-enumerable/
    Interfaces/
      Enumerators/
        interface I_ForwardEnumerator: IsValid, MoveNext, Reset, TryGet, TryGetTo
        interface I_KeyValueForwardEnumerator: Key
      interface I_Enumerable: GetEnumerator
      interface I_KeyValueEnumerable: GetKeyValueEnumerator
  mobject-errors/
    Errors/
      function block Error [ST]: OnSerialize, Accept, ErrorType, IsSameAs, Message, SerializeWith
      function block NullError [ST]: ErrorType, Message, SerializeWith
    Interfaces/
      interface I_Error: Accept, ErrorType, IsSameAs, Message
      interface I_ErrorVisitor: VisitError
  mobject-events/
    _Internal/
      EventHandlerItem/
        function block EventHandlerItem [ST]: FB_init, Emit, EqualTo, Next, Previous
        function block EventHandlerItemOnceOnly [ST]: FB_init, Emit
        interface I_EventHandlerItem: Emit, EqualTo, Next, Previous
    EventEmitter/
      function block EventEmitter [ST]: FB_exit, DisposeAllEventHandlerItems, DisposeEventHandlerItem, FindEventHandlerItem, InsertEventHandlerItem, RemoveEventHandlerItemFromCollection, Clear, Emit, OffEvent, OnceEvent, OnEvent
    Interfaces/
      interface I_Event
      interface I_EventEmitter: OffEvent, OnceEvent, OnEvent
      interface I_EventHandler: HandleEvent
      interface I_EventTarget: Emit
  mobject-json/
    _Internal/
      Events/
        function block JsonDeserializerChangedEvent [ST]
        function block JsonDeserializerDisposedEvent [ST]
        function block JsonDeserializerEvent [ST]: FB_init, Target
      JsonDeserializerForwardEnumerator/
        function block JsonDeserializerArrayForwardEnumerator [ST]: FB_init, FB_exit, CreateDeserializer, Initialize, UpdateCurrentDeserializer, Current, HandleEvent, Index, IsValid, MoveNext
        function block JsonDeserializerNullArrayForwardEnumerator [ST]: FB_init, FB_exit, Current, HandleEvent, Index, IsValid, MoveNext
        function block JsonDeserializerNullObjectForwardEnumerator [ST]: FB_init, FB_exit, Current, HandleEvent, IsValid, Key, MoveNext
        function block JsonDeserializerObjectForwardEnumerator [ST]: FB_init, FB_exit, CreateDeserializer, Initialize, UpdateCurrentDeserializer, Current, HandleEvent, IsValid, Key, MoveNext
      JsonDeserializerNode/
        function block JsonDeserializerNode [ST]: FB_init, CreateArrayForwardEnumerator, CreateDeserializer, CreateObjectForwardEnumerator, TryGetMember, TryReadBool, TryReadNumber, TryReadString, TryReadStringEx, Clone, Dispose, GetArray, GetArrayEnumerator, GetElementByIndex, GetKeyArray, GetKeyObject, GetObject, GetObjectEnumerator, GetValue, TryDeserializeKeyToObject, TryDeserializeToObject, TryGetBase64, TryGetBool, TryGetByte, TryGetDateTime, TryGetDcTime, TryGetDint, TryGetDword, TryGetElementByIndex, TryGetFileTime, TryGetHexAsBytes, TryGetInt, TryGetKeyBase64, TryGetKeyBool, TryGetKeyByte, TryGetKeyDateTime, TryGetKeyDcTime, TryGetKeyDint, TryGetKeyDword, TryGetKeyFileTime, TryGetKeyHexAsBytes, TryGetKeyInt, TryGetKeyLint, TryGetKeyLreal, TryGetKeyLtime, TryGetKeyLword, TryGetKeyReal, TryGetKeySint, TryGetKeyString, TryGetKeyStringEx, TryGetKeyTime, TryGetKeyTod, TryGetKeyUdint, TryGetKeyUint, TryGetKeyUlint, TryGetKeyUsint, TryGetKeyWord, TryGetLint, TryGetLreal, TryGetLtime, TryGetLword, TryGetReal, TryGetSint, TryGetString, TryGetStringEx, TryGetTime, TryGetTod, TryGetUdint, TryGetUint, TryGetUlint, TryGetUsint, TryGetWord
        function block JsonDeserializerNullNode [ST]: FB_init, CreateNullArrayEnumerator, CreateNullObjectEnumerator, Clone, GetArray, GetArrayEnumerator, GetElementByIndex, GetKeyArray, GetKeyObject, GetObject, GetObjectEnumerator, TryDeserializeKeyToObject, TryDeserializeToObject, TryGetBase64, TryGetBool, TryGetByte, TryGetDateTime, TryGetDcTime, TryGetDint, TryGetDword, TryGetElementByIndex, TryGetFileTime, TryGetHexAsBytes, TryGetInt, TryGetKeyBase64, TryGetKeyBool, TryGetKeyByte, TryGetKeyDateTime, TryGetKeyDcTime, TryGetKeyDint, TryGetKeyDword, TryGetKeyFileTime, TryGetKeyHexAsBytes, TryGetKeyInt, TryGetKeyLint, TryGetKeyLreal, TryGetKeyLtime, TryGetKeyLword, TryGetKeyReal, TryGetKeySint, TryGetKeyString, TryGetKeyStringEx, TryGetKeyTime, TryGetKeyTod, TryGetKeyUdint, TryGetKeyUint, TryGetKeyUlint, TryGetKeyUsint, TryGetKeyWord, TryGetLint, TryGetLreal, TryGetLtime, TryGetLword, TryGetReal, TryGetSint, TryGetString, TryGetStringEx, TryGetTime, TryGetTod, TryGetUdint, TryGetUint, TryGetUlint, TryGetUsint, TryGetWord
      JsonPathSyntaxParser/
        function block JsonPathSyntaxParser [ST]: Parse
      JsonPathVisitor/
        interface I_JsonPathVisitor: ArrayIndexFound, EndOfParse, InvalidSyntaxFound, PropertyFound, StartOfParse
        function block JsonDomCreator [ST]: FB_init, PadStartOfArray, ArrayIndexFound, CurrentNode, EndOfParse, InvalidSyntaxFound, PropertyFound, StartOfParse
        function block JsonDomNavigator [ST]: FB_init, ArrayIndexFound, CurrentNode, EndOfParse, InvalidSyntaxFound, PropertyFound, StartOfParse
    JsonDeserializer/
      Events/
        interface I_JsonDeserializerChangedEvent: Target
        interface I_JsonDeserializerDisposedEvent: Target
      interface I_JsonDeserializer
      function block JsonDeserializer [ST]: FB_exit, CreateDeserializer, EmitChangedEvent, EmitDisposedEvent, Clone, GetArray, GetArrayEnumerator, GetElementByIndex, GetKeyArray, GetKeyObject, GetObject, GetObjectEnumerator, OffEvent, OnceEvent, OnEvent, Reset, TryDeserializeKeyToObject, TryDeserializeToObject, TryGetBase64, TryGetBool, TryGetByte, TryGetDateTime, TryGetDcTime, TryGetDint, TryGetDword, TryGetElementByIndex, TryGetFileTime, TryGetHexAsBytes, TryGetInt, TryGetKeyBase64, TryGetKeyBool, TryGetKeyByte, TryGetKeyDateTime, TryGetKeyDcTime, TryGetKeyDint, TryGetKeyDword, TryGetKeyFileTime, TryGetKeyHexAsBytes, TryGetKeyInt, TryGetKeyLint, TryGetKeyLreal, TryGetKeyLtime, TryGetKeyLword, TryGetKeyReal, TryGetKeySint, TryGetKeyString, TryGetKeyStringEx, TryGetKeyTime, TryGetKeyTod, TryGetKeyUdint, TryGetKeyUint, TryGetKeyUlint, TryGetKeyUsint, TryGetKeyWord, TryGetLint, TryGetLreal, TryGetLtime, TryGetLword, TryGetReal, TryGetSint, TryGetString, TryGetStringEx, TryGetTime, TryGetTod, TryGetUdint, TryGetUint, TryGetUlint, TryGetUsint, TryGetWord, TryLoad
    JsonDomParser/
      function block JsonDomParser [ST]: TrySetBool, TrySetDouble, TrySetInt, TrySetInt64, TrySetString, TrySetUint, TrySetUint64, TryLocate, TryModify, TryRead, TryWrite
    JsonSerializer/
      function block JsonSerializer [ST]: FB_exit, AddBase64, AddBool, AddByte, AddBytesAsHex, AddDateTime, AddDcTime, AddDint, AddDword, AddFileTime, AddInt, AddKey, AddKeyBase64, AddKeyBool, AddKeyByte, AddKeyBytesAsHex, AddKeyDateTime, AddKeyDcTime, AddKeyDint, AddKeyDword, AddKeyFileTime, AddKeyInt, AddKeyLint, AddKeyLreal, AddKeyLtime, AddKeyLword, AddKeyNull, AddKeyObject, AddKeyRawJson, AddKeyReal, AddKeySint, AddKeyString, AddKeyStringByRef, AddKeyTime, AddKeyTod, AddKeyUdint, AddKeyUint, AddKeyUlint, AddKeyUsint, AddKeyWord, AddLint, AddLreal, AddLtime, AddLword, AddNull, AddObject, AddRawJson, AddReal, AddSint, AddString, AddStringByRef, AddTime, AddTod, AddUdint, AddUint, AddUlint, AddUsint, AddWord, Clone, EndArray, EndObject, GetSerializedDataLength, Reset, StartArray, StartObject, TryCopySerializedData, TryGetSerializedData
  mobject-serialization/
    Interfaces/
      interface I_Serializable: SerializeWith
      interface I_Serializer: AddBase64, AddBool, AddByte, AddBytesAsHex, AddDateTime, AddDcTime, AddDint, AddDword, AddFileTime, AddInt, AddKey, AddKeyBase64, AddKeyBool, AddKeyByte, AddKeyBytesAsHex, AddKeyDateTime, AddKeyDcTime, AddKeyDint, AddKeyDword, AddKeyFileTime, AddKeyInt, AddKeyLint, AddKeyLreal, AddKeyLtime, AddKeyLword, AddKeyNull, AddKeyObject, AddKeyReal, AddKeySint, AddKeyString, AddKeyStringByRef, AddKeyTime, AddKeyTod, AddKeyUdint, AddKeyUint, AddKeyUlint, AddKeyUsint, AddKeyWord, AddLint, AddLreal, AddLtime, AddLword, AddNull, AddObject, AddReal, AddSint, AddString, AddStringByRef, AddTime, AddTod, AddUdint, AddUint, AddUlint, AddUsint, AddWord, Clone, EndArray, EndObject, GetSerializedDataLength, Reset, StartArray, StartObject, TryCopySerializedData, TryGetSerializedData
  mobject-server/
    _Internal/
      AsyncResponse/
        HeaderAccessor/
          interface I_AsyncResponseHeaderAccessor: TryGetResponseIdFromRequest, TryGetSessionIdFromRequest, TryGetSessionIdFromResponse
        Manager/
          function block AsyncResponseManager [ST]: FB_init, CreateAsyncResponseSessionData, CreateAsyncResponseSessionDataProxy, TryConvertResponseToAsyncResponseSessionData, TryHandleIncomingRequest
          interface I_AsyncResponseManager: TryConvertResponseToAsyncResponseSessionData, TryHandleIncomingRequest
        Middleware/
          function block AsyncResponseMiddleware [ST]: FB_init, Handle
        Proxy/
          function block AsyncResponseSessionDataProxy [ST]: FB_init, TryGetAsyncResponseSessionData, Error, HasExpired, IsPending, Success, SuccessWithPayload, SuggestedRetryDelayInMs, TryUpdateServerResponse
        SessionData/
          function block AsyncResponseSessionData [ST]: FB_init, FB_exit, CopyPayloadData, DeletePayloadData, Error, HasExpired, IsPending, Success, SuccessWithPayload, SuggestedRetryDelayInMs, TryUpdateServerResponse
          interface I_AsyncResponseSessionData: Error, HasExpired, IsPending, Success, SuccessWithPayload, SuggestedRetryDelayInMs, TryUpdateServerResponse
      ChunkedRequests/
        ChunkedRequest/
          function block ChunkedRequest [ST]: FB_init, CreatedTimestamp, Header, PayloadAddress, PayloadSizeInBytes
        HeaderAccessor/
          interface I_ChunkedRequestsHeaderAccessor: TryGetChunkSequenceFromRequest, TryGetChunkTotalFromRequest, TryGetHasMoreChunksFromRequest, TryGetRequestIdFromRequest, TryGetSessionIdFromRequest
        Manager/
          function block ChunkedRequestsManager [ST]: FB_init, CreateChunkedRequestData, TryHandleIncomingRequest
          interface I_ChunkedRequestsManager: TryHandleIncomingRequest
        Middleware/
          function block ChunkedRequestsMiddleware [ST]: FB_init, Handle
        SessionData/
          function block ChunkedRequestData [ST]: FB_init, FB_exit, CreateBuffer, DestroyBuffer, IsComplete, PayloadAddress, PayloadSizeInBytes, TryAddChunkedPayload
          interface I_ChunkedRequestData: IsComplete, PayloadAddress, PayloadSizeInBytes, TryAddChunkedPayload
      ChunkedResponses/
        HeaderAccessor/
          interface I_ChunkedResponseHeaderAccessor: TryGetResponseIdFromRequest, TryGetSessionIdFromRequest, TryGetSessionIdFromResponse, UpdateResponseWithHasMoreChunks
        Manager/
          function block ChunkedResponseManager [ST]: FB_init, CreateChunkedResponseData, HandleSuccessWithPayload, TryHandleIncomingRequest
          interface I_ChunkedResponseManager: HandleSuccessWithPayload, TryHandleIncomingRequest
        Middleware/
          function block ChunkedResponsesMiddleware [ST]: FB_init, Handle
        ServerResponse/
          function block ChunkableServerResponse [ST]: FB_init, Accepted, Busy, Error, Header, HeadersSent, Pending, Success, SuccessWithPayload
        SessionData/
          function block ChunkedResponseData [ST]: FB_init, FB_exit, StoreData, SendComplete, SendNextChunk, SizeRemaining
          interface I_ChunkedResponseData: SendComplete, SendNextChunk, SizeRemaining
      Followup/
        Middleware/
          function block ResponseIdGuardMiddleware [ST]: FB_init, Handle
      Header/
        function block Header [ST]: FB_init, FB_exit, ToString, TryGetField, TryWriteField
        interface I_Header: ToString, TryGetField, TryWriteField
      HeaderAccessor/
        function block HeaderAccessor [ST]: ContentType_Json, HeaderKey_Accept, HeaderKey_ChunkSequence, HeaderKey_ChunkTotal, HeaderKey_ContentType, HeaderKey_ErrorCode, HeaderKey_ErrorMessage, HeaderKey_HasMoreChunks, HeaderKey_MethodName, HeaderKey_RequestId, HeaderKey_ResponseId, HeaderKey_RetryDelay, HeaderKey_SessionId, HeaderKey_Status, HeaderKey_Type, StatusValue_Accepted, StatusValue_Busy, StatusValue_Error, StatusValue_Pending, StatusValue_Success, TryGetAcceptResponseFormatFromRequest, TryGetChunkSequenceFromRequest, TryGetChunkTotalFromRequest, TryGetContentTypeFromRequest, TryGetHasMoreChunksFromRequest, TryGetMethodNameFromRequest, TryGetRequestIdFromRequest, TryGetResponseIdFromRequest, TryGetSessionIdFromRequest, TryGetSessionIdFromResponse, TryGetTypeFromRequest, UpdateRequestWithSessionId, UpdateResponseWithAccepted, UpdateResponseWithBusy, UpdateResponseWithError, UpdateResponseWithHasMoreChunks, UpdateResponseWithPending, UpdateResponseWithSessionId, UpdateResponseWithSuccess
      Middleware/
        Base/
          function block MiddlewareBase [ST]: Next, Handle, NextMiddleware
        Interface/
          interface I_Middleware: Handle, NextMiddleware
        Stack/
          function block MiddlewareStack [ST]: Handle, Use
      Request/
        Interface/
          interface I_Request: CreatedTimestamp, Header, PayloadAddress, PayloadSizeInBytes
        function block Request [ST]: FB_init, CreatedTimestamp, Header, PayloadAddress, PayloadSizeInBytes
      ResponseId/
        Interface/
          interface I_ResponseIdGenerator: Generate
        function block SequentialResponseIdGenerator [ST]: Generate
      RPC/
        AsyncRpcCall/
          function block AsyncRpcCall [ST]: FB_init, FB_exit, Call
          interface I_AsyncRpcCall: Call
        AsyncRpcCallQueue/
          function block AsyncRpcCallQueue [ST]: FB_exit, CreateCall, DisposeAll, CyclicCall, TryAddRpcCall
          interface I_AsyncRpcCallQueue: TryAddRpcCall
        Handlers/
          function block AsynchronousRpcHandlers [ST]: HasHandlers, RegisterHandler, TryGetByMethodName
          interface I_AsynchronousRpcHandlers: HasHandlers, TryGetByMethodName
          interface I_HostAsynchronousRpcHandlers: RegisterHandler
          interface I_HostSynchronousRpcHandlers: RegisterHandler
          interface I_SynchronousRpcHandlers: HasHandlers, TryGetByMethodName
          function block SynchronousRpcHandlers [ST]: HasHandlers, RegisterHandler, TryGetByMethodName
        HeaderAccessor/
          interface I_RpcHeaderAccessor: ContentType_Json, TryGetAcceptResponseFormatFromRequest, TryGetContentTypeFromRequest, TryGetMethodNameFromRequest, TryGetTypeFromRequest
        Manager/
          interface I_RpcManager: TryHandleIncomingRequest
          function block RpcManager [ST]: FB_init, HandleAsyncRpcRequest, HandleSyncRpcRequest, TryCreateAsynchronousRpcResponse, TryCreateDeserializer, TryCreateSerializer, TryCreateSynchronousRpcResponse, TryHandleIncomingRequest
        Middleware/
          function block RpcMiddleware [ST]: FB_init, Handle
        RegisteredRpcApis/
          function block RegisteredRpcApis [ST]: FB_exit, CreateEnumerator, CyclicCall, HasRegisteredRpcApis, RegisterRpcApi
        Response/
          Async/
            function block AsynchronousRpcResponse [ST]: FB_init, FB_exit, SendSuccessResponseUsingSeralizer, CompleteWithBase64, CompleteWithBool, CompleteWithBytesAsHex, CompleteWithDateTime, CompleteWithDcTime, CompleteWithDint, CompleteWithFileTime, CompleteWithLint, CompleteWithLreal, CompleteWithNull, CompleteWithObject, CompleteWithReal, CompleteWithSerializer, CompleteWithString, CompleteWithUdint, CompleteWithUlint, GetSerializer, RejectWithError
            interface I_AsynchronousRpcResponse: CompleteWithBase64, CompleteWithBool, CompleteWithBytesAsHex, CompleteWithDateTime, CompleteWithDcTime, CompleteWithDint, CompleteWithFileTime, CompleteWithLint, CompleteWithLreal, CompleteWithNull, CompleteWithObject, CompleteWithReal, CompleteWithSerializer, CompleteWithString, CompleteWithUdint, CompleteWithUlint, GetSerializer, RejectWithError
          Factory/
            function block AsynchronousRpcResponseFactory [ST]: FB_init, TryCreate
            interface I_AsynchronousRpcResponseFactory: TryCreate
          Sync/
            interface I_SynchronousRpcResponse: CompleteWithBase64, CompleteWithBool, CompleteWithBytesAsHex, CompleteWithDateTime, CompleteWithDcTime, CompleteWithDint, CompleteWithFileTime, CompleteWithLint, CompleteWithLreal, CompleteWithNull, CompleteWithObject, CompleteWithReal, CompleteWithSerializer, CompleteWithString, CompleteWithUdint, CompleteWithUlint, GetSerializer, RejectWithError, TryMakeAsynchronous
            function block SynchronousRpcResponse [ST]: FB_init, FB_exit, SendSuccessResponseUsingSeralizer, CompleteWithBase64, CompleteWithBool, CompleteWithBytesAsHex, CompleteWithDateTime, CompleteWithDcTime, CompleteWithDint, CompleteWithFileTime, CompleteWithLint, CompleteWithLreal, CompleteWithNull, CompleteWithObject, CompleteWithReal, CompleteWithSerializer, CompleteWithString, CompleteWithUdint, CompleteWithUlint, GetSerializer, RejectWithError, TryMakeAsynchronous
      ServerResponse/
        Data/
          data type ResponseData
        HeaderAccessor/
          interface I_ServerResponseHeaderAccessor: UpdateResponseWithAccepted, UpdateResponseWithBusy, UpdateResponseWithError, UpdateResponseWithPending, UpdateResponseWithSuccess
        Interface/
          interface I_ServerResponse: Accepted, Busy, Error, Header, HeadersSent, Pending, Success, SuccessWithPayload
        function block ServerResponse [ST]: FB_init, CompleteResponseWithoutPayload, CompleteResponseWithPayload, Accepted, Busy, Error, Header, HeadersSent, Pending, Success, SuccessWithPayload, TryGetData
      Sessions/
        HeaderAccessor/
          interface I_SessionHeaderAccessor: TryGetResponseIdFromRequest, TryGetSessionIdFromRequest, UpdateRequestWithSessionId, UpdateResponseWithSessionId
        Manager/
          interface I_SessionManager: CreateSession, DisposeAllSessions, IsValidSession, RefreshSession
          function block SessionManager [ST]: FB_init, FB_exit, CheckForExpiredSessions, CreateNewSession, CreateSession, CyclicCall, DisposeAllSessions, DisposeSession, DisposeSessionDataById, IsValidSession, RefreshSession, SessionCount, TryRetrieveSessionDataById, TryStoreSessionDataById
        Middleware/
          function block SessionsMiddleware [ST]: FB_init, Handle
        Session/
          interface I_Session: AddOrUpdateStorage, DisposeAllDataFromStorage, DisposeDataFromStorage, Id, LastAccessedTimestamp, Refresh, TryGetDataFromStorage
          function block Session [ST]: FB_init, FB_exit, AddOrUpdateStorage, DisposeAllDataFromStorage, DisposeDataFromStorage, Id, LastAccessedTimestamp, Refresh, TryGetDataFromStorage
        SessionData/
          interface I_SessionData
        SessionId/
          interface I_SessionIdGenerator: Generate
          function block SequentialSessionIdGenerator [ST]: Generate
        Storage/
          interface I_SessionStorage: DisposeSessionDataById, TryRetrieveSessionDataById, TryStoreSessionDataById
      TimeStamp/
        interface I_Timestamp: IsDurationElapsed, TimeSince
        function block SystemTimestamp [ST]: FB_init, IsDurationElapsed, SetNow, TimeSince
    GVLs/
      global variables ServerConfiguration
    RpcApi/
      interface I_RpcApi: CyclicCall, RegisterAsynchronousRpcHandlersWith, RegisterSynchronousRpcHandlersWith
    RpcHandler/
      Examples/
        function block AsyncConcatStringRpcHandler [ST]: Handle
        function block ConcatStringRpcHandler [ST]: Handle
      interface I_AsynchronousRpcHandler: Handle
      interface I_SynchronousRpcHandler: Handle
    RpcServer/
      interface I_RpcServer: GetConfiguredHeaderSize, GetConfiguredPayloadSize, HandleRequest, RegisterApi, RegisterAsynchronousRpcHandler, RegisterSynchronousRpcHandler
      function block RpcServer [ST]: FB_init, CyclicCall, GetConfiguredHeaderSize, GetConfiguredPayloadSize, HandleRequest, RegisterApi, RegisterAsynchronousRpcHandler, RegisterSynchronousRpcHandler, SessionCount, Use
*)

// mobject-server/_Internal/ServerResponse/Data/ResponseData
TYPE ResponseData : 
STRUCT
	Header : STRING(ServerConfiguration.HEADER_STRING_SIZE);
	Payload : STRING(ServerConfiguration.PAYLOAD_STRING_SIZE);
END_STRUCT
END_TYPE

// mobject-constants/DatatypeLimits
{attribute 'qualified_only'}
VAR_GLOBAL CONSTANT
                
	// Boolean
	BOOL_MIN_VALUE : BOOL := FALSE;
	BOOL_MAX_VALUE : BOOL := TRUE;
	
	// Integer Datatypes
	BYTE_MIN_VALUE : BYTE := BYTE#0;
	BYTE_MAX_VALUE : BYTE := BYTE#255;
	WORD_MIN_VALUE : WORD := WORD#0;
	WORD_MAX_VALUE : WORD := WORD#65535;
	DWORD_MIN_VALUE : DWORD := DWORD#0;
	DWORD_MAX_VALUE : DWORD := DWORD#4294967295;
	LWORD_MIN_VALUE : LWORD := LWORD#0;
	LWORD_MAX_VALUE : LWORD := LWORD#18446744073709551615;
	SINT_MIN_VALUE : SINT := SINT#-128;
	SINT_MAX_VALUE : SINT := SINT#127;
	USINT_MIN_VALUE : USINT := USINT#0;
	USINT_MAX_VALUE : USINT := USINT#255;
	INT_MIN_VALUE : INT := INT#-32768;
	INT_MAX_VALUE : INT := INT#32767;
	UINT_MIN_VALUE : UINT := UINT#0;
	UINT_MAX_VALUE : UINT := UINT#65535;
	DINT_MIN_VALUE : DINT := DINT#-2147483648;
	DINT_MAX_VALUE : DINT := DINT#2147483647;
	UDINT_MIN_VALUE : UDINT := UDINT#0;
	UDINT_MAX_VALUE : UDINT := UDINT#4294967295;
	LINT_MIN_VALUE : LINT := LINT#-9223372036854775808;
	LINT_MAX_VALUE : LINT := LINT#9223372036854775807;
	ULINT_MIN_VALUE : ULINT := ULINT#0;
	ULINT_MAX_VALUE : ULINT := ULINT#18446744073709551615;
	
	// Floating-point types
	REAL_MAX_VALUE : REAL := REAL#3.402823E+38; // Largest positive REAL number
	REAL_MIN_VALUE : REAL := REAL#-3.402823E+38; // Largest negative REAL number
	REAL_POSITIVE_MIN_VALUE : REAL := REAL#1.0E-44; // Smallest positive REAL number
	REAL_NEGATIVE_MIN_VALUE : REAL := REAL#-1.0E-44; // Smallest negative REAL number
	LREAL_MAX_VALUE : LREAL := LREAL#1.7976931348623157E+308; // Largest positive LREAL number
	LREAL_MIN_VALUE : LREAL := LREAL#-1.7976931348623157E+308; // Largest negative LREAL number
	LREAL_POSITIVE_MIN_VALUE : LREAL := LREAL#4.94065645841247E-324; // Smallest positive LREAL number
	LREAL_NEGATIVE_MIN_VALUE : LREAL := LREAL#-4.94065645841247E-324; // Smallest negative LREAL number
	
	// Time Datatypes
	TIME_MIN_VALUE : TIME := T#0MS;
	TIME_MAX_VALUE : TIME := T#49D17H2M47S295MS;
	
	// Date
	DATE_MIN_VALUE : DATE := DATE#1970-1-1;
	DATE_MAX_VALUE : DATE := DATE#2106-2-7;
	DT_MIN_VALUE : DATE_AND_TIME := DATE_AND_TIME#1970-1-1-0:0:0;
	DT_MAX_VALUE : DATE_AND_TIME := DATE_AND_TIME#2106-02-07-06:28:15;
	TOD_MIN_VALUE : TIME_OF_DAY := TIME_OF_DAY#0:0:0;
	TOD_MAX_VALUE : TIME_OF_DAY := TIME_OF_DAY#23:59:59.999;
	
	// -----------------------------------------------------------------------------
	
	// Limits of BYTE used for conversions
	MAX_VALUE_OF_BYTE_WHICH_CAN_BE_HELD_IN_A_SINT : BYTE := BYTE#127;
	
	// Limits of WORD used for conversions
	MAX_VALUE_OF_WORD_WHICH_CAN_BE_HELD_IN_A_BYTE : WORD := WORD#255;
	MAX_VALUE_OF_WORD_WHICH_CAN_BE_HELD_IN_A_SINT : WORD := WORD#127;
	MAX_VALUE_OF_WORD_WHICH_CAN_BE_HELD_IN_A_INT : WORD := WORD#32767;
	MAX_VALUE_OF_WORD_WHICH_CAN_BE_HELD_IN_A_USINT : WORD := WORD#255;
	
	// Limits of DWORD used for conversions
	MAX_VALUE_OF_DWORD_WHICH_CAN_BE_HELD_IN_A_BYTE : DWORD := DWORD#255;
	MAX_VALUE_OF_DWORD_WHICH_CAN_BE_HELD_IN_A_WORD : DWORD := DWORD#65535;
	MAX_VALUE_OF_DWORD_WHICH_CAN_BE_HELD_IN_A_SINT : DWORD := DWORD#127;
	MAX_VALUE_OF_DWORD_WHICH_CAN_BE_HELD_IN_A_INT : DWORD := DWORD#32767;
	MAX_VALUE_OF_DWORD_WHICH_CAN_BE_HELD_IN_A_DINT : DWORD := DWORD#2147483647;
	MAX_VALUE_OF_DWORD_WHICH_CAN_BE_HELD_IN_A_USINT : DWORD := DWORD#255;
	MAX_VALUE_OF_DWORD_WHICH_CAN_BE_HELD_IN_A_UINT : DWORD := DWORD#65535;
	MAX_VALUE_OF_DWORD_WHICH_CAN_BE_HELD_IN_A_TOD : DWORD := DWORD#86399999;
	
	// Limits of LWORD used for conversions
	MAX_VALUE_OF_LWORD_WHICH_CAN_BE_HELD_IN_A_BYTE : LWORD := LWORD#255;
	MAX_VALUE_OF_LWORD_WHICH_CAN_BE_HELD_IN_A_WORD : LWORD := LWORD#65535;
	MAX_VALUE_OF_LWORD_WHICH_CAN_BE_HELD_IN_A_DWORD : LWORD := LWORD#4294967295;
	MAX_VALUE_OF_LWORD_WHICH_CAN_BE_HELD_IN_A_SINT : LWORD := LWORD#127;
	MAX_VALUE_OF_LWORD_WHICH_CAN_BE_HELD_IN_A_INT : LWORD := LWORD#32767;
	MAX_VALUE_OF_LWORD_WHICH_CAN_BE_HELD_IN_A_DINT : LWORD := LWORD#2147483647;
	MAX_VALUE_OF_LWORD_WHICH_CAN_BE_HELD_IN_A_LINT : LWORD := LWORD#9223372036854775807;
	MAX_VALUE_OF_LWORD_WHICH_CAN_BE_HELD_IN_A_USINT : LWORD := LWORD#255;
	MAX_VALUE_OF_LWORD_WHICH_CAN_BE_HELD_IN_A_UINT : LWORD := LWORD#65535;
	MAX_VALUE_OF_LWORD_WHICH_CAN_BE_HELD_IN_A_UDINT : LWORD := LWORD#4294967295;
	MAX_VALUE_OF_LWORD_WHICH_CAN_BE_HELD_IN_A_TIME : LWORD := LWORD#4294967295;
	MAX_VALUE_OF_LWORD_WHICH_CAN_BE_HELD_IN_A_TOD : LWORD := LWORD#86399999;
	MAX_VALUE_OF_LWORD_WHICH_CAN_BE_HELD_IN_A_DATE : LWORD := LWORD#4294967295;
	MAX_VALUE_OF_LWORD_WHICH_CAN_BE_HELD_IN_A_DT : LWORD := LWORD#4294967295;
	
	// Limits of SINT used for conversions
	MIN_VALUE_OF_SINT_WHICH_CAN_BE_HELD_IN_A_BYTE : SINT := SINT#0;
	MIN_VALUE_OF_SINT_WHICH_CAN_BE_HELD_IN_A_WORD : SINT := SINT#0;
	MIN_VALUE_OF_SINT_WHICH_CAN_BE_HELD_IN_A_DWORD : SINT := SINT#0;
	MIN_VALUE_OF_SINT_WHICH_CAN_BE_HELD_IN_A_LWORD : SINT := SINT#0;
	MIN_VALUE_OF_SINT_WHICH_CAN_BE_HELD_IN_A_USINT : SINT := SINT#0;
	MIN_VALUE_OF_SINT_WHICH_CAN_BE_HELD_IN_A_UINT : SINT := SINT#0;
	MIN_VALUE_OF_SINT_WHICH_CAN_BE_HELD_IN_A_UDINT : SINT := SINT#0;
	MIN_VALUE_OF_SINT_WHICH_CAN_BE_HELD_IN_A_ULINT : SINT := SINT#0;
	MIN_VALUE_OF_SINT_WHICH_CAN_BE_HELD_IN_A_TIME : SINT := SINT#0;
	MIN_VALUE_OF_SINT_WHICH_CAN_BE_HELD_IN_A_TOD : SINT := SINT#0;
	MIN_VALUE_OF_SINT_WHICH_CAN_BE_HELD_IN_A_DATE : SINT := SINT#0;
	MIN_VALUE_OF_SINT_WHICH_CAN_BE_HELD_IN_A_DT : SINT := SINT#0;
	
	// Limits of INT used for conversions
	MIN_VALUE_OF_INT_WHICH_CAN_BE_HELD_IN_A_BYTE : INT := INT#0;
	MAX_VALUE_OF_INT_WHICH_CAN_BE_HELD_IN_A_BYTE : INT := INT#255;
	MIN_VALUE_OF_INT_WHICH_CAN_BE_HELD_IN_A_WORD : INT := INT#0;
	MIN_VALUE_OF_INT_WHICH_CAN_BE_HELD_IN_A_DWORD : INT := INT#0;
	MIN_VALUE_OF_INT_WHICH_CAN_BE_HELD_IN_A_LWORD : INT := INT#0;
	MIN_VALUE_OF_INT_WHICH_CAN_BE_HELD_IN_A_SINT : INT := INT#-128;
	MAX_VALUE_OF_INT_WHICH_CAN_BE_HELD_IN_A_SINT : INT := INT#127;
	MIN_VALUE_OF_INT_WHICH_CAN_BE_HELD_IN_A_USINT : INT := INT#0;
	MAX_VALUE_OF_INT_WHICH_CAN_BE_HELD_IN_A_USINT : INT := INT#255;
	MIN_VALUE_OF_INT_WHICH_CAN_BE_HELD_IN_A_UINT : INT := INT#0;
	MIN_VALUE_OF_INT_WHICH_CAN_BE_HELD_IN_A_UDINT : INT := INT#0;
	MIN_VALUE_OF_INT_WHICH_CAN_BE_HELD_IN_A_ULINT : INT := INT#0;
	MIN_VALUE_OF_INT_WHICH_CAN_BE_HELD_IN_A_TIME : INT := INT#0;
	MIN_VALUE_OF_INT_WHICH_CAN_BE_HELD_IN_A_TOD : INT := INT#0;
	MIN_VALUE_OF_INT_WHICH_CAN_BE_HELD_IN_A_DATE : INT := INT#0;
	MIN_VALUE_OF_INT_WHICH_CAN_BE_HELD_IN_A_DT : INT := INT#0;
	
	// Limits of DINT used for conversions
	MIN_VALUE_OF_DINT_WHICH_CAN_BE_HELD_IN_A_BYTE : DINT := DINT#0;
	MAX_VALUE_OF_DINT_WHICH_CAN_BE_HELD_IN_A_BYTE : DINT := DINT#255;
	MIN_VALUE_OF_DINT_WHICH_CAN_BE_HELD_IN_A_WORD : DINT := DINT#0;
	MAX_VALUE_OF_DINT_WHICH_CAN_BE_HELD_IN_A_WORD : DINT := DINT#65535;
	MIN_VALUE_OF_DINT_WHICH_CAN_BE_HELD_IN_A_DWORD : DINT := DINT#0;
	MIN_VALUE_OF_DINT_WHICH_CAN_BE_HELD_IN_A_LWORD : DINT := DINT#0;
	MIN_VALUE_OF_DINT_WHICH_CAN_BE_HELD_IN_A_SINT : DINT := DINT#-128;
	MAX_VALUE_OF_DINT_WHICH_CAN_BE_HELD_IN_A_SINT : DINT := DINT#127;
	MIN_VALUE_OF_DINT_WHICH_CAN_BE_HELD_IN_A_INT : DINT := DINT#-32768;
	MAX_VALUE_OF_DINT_WHICH_CAN_BE_HELD_IN_A_INT : DINT := DINT#32767;
	MIN_VALUE_OF_DINT_WHICH_CAN_BE_HELD_IN_A_USINT : DINT := DINT#0;
	MAX_VALUE_OF_DINT_WHICH_CAN_BE_HELD_IN_A_USINT : DINT := DINT#255;
	MIN_VALUE_OF_DINT_WHICH_CAN_BE_HELD_IN_A_UINT : DINT := DINT#0;
	MAX_VALUE_OF_DINT_WHICH_CAN_BE_HELD_IN_A_UINT : DINT := DINT#65535;
	MIN_VALUE_OF_DINT_WHICH_CAN_BE_HELD_IN_A_UDINT : DINT := DINT#0;
	MIN_VALUE_OF_DINT_WHICH_CAN_BE_HELD_IN_A_ULINT : DINT := DINT#0;
	MIN_VALUE_OF_DINT_WHICH_CAN_BE_HELD_IN_A_TIME : DINT := DINT#0;
	MIN_VALUE_OF_DINT_WHICH_CAN_BE_HELD_IN_A_TOD : DINT := DINT#0;
	MAX_VALUE_OF_DINT_WHICH_CAN_BE_HELD_IN_A_TOD : DINT := DINT#86399999;
	MIN_VALUE_OF_DINT_WHICH_CAN_BE_HELD_IN_A_DATE : DINT := DINT#0;
	MIN_VALUE_OF_DINT_WHICH_CAN_BE_HELD_IN_A_DT : DINT := DINT#0;
	
	// Limits of LINT used for conversions
	MIN_VALUE_OF_LINT_WHICH_CAN_BE_HELD_IN_A_BYTE : LINT := LINT#0;
	MAX_VALUE_OF_LINT_WHICH_CAN_BE_HELD_IN_A_BYTE : LINT := LINT#255;
	MIN_VALUE_OF_LINT_WHICH_CAN_BE_HELD_IN_A_WORD : LINT := LINT#0;
	MAX_VALUE_OF_LINT_WHICH_CAN_BE_HELD_IN_A_WORD : LINT := LINT#65535;
	MIN_VALUE_OF_LINT_WHICH_CAN_BE_HELD_IN_A_DWORD : LINT := LINT#0;
	MAX_VALUE_OF_LINT_WHICH_CAN_BE_HELD_IN_A_DWORD : LINT := LINT#4294967295;
	MIN_VALUE_OF_LINT_WHICH_CAN_BE_HELD_IN_A_LWORD : LINT := LINT#0;
	MIN_VALUE_OF_LINT_WHICH_CAN_BE_HELD_IN_A_SINT : LINT := LINT#-128;
	MAX_VALUE_OF_LINT_WHICH_CAN_BE_HELD_IN_A_SINT : LINT := LINT#127;
	MIN_VALUE_OF_LINT_WHICH_CAN_BE_HELD_IN_A_INT : LINT := LINT#-32768;
	MAX_VALUE_OF_LINT_WHICH_CAN_BE_HELD_IN_A_INT : LINT := LINT#32767;
	MIN_VALUE_OF_LINT_WHICH_CAN_BE_HELD_IN_A_DINT : LINT := LINT#-2147483648;
	MAX_VALUE_OF_LINT_WHICH_CAN_BE_HELD_IN_A_DINT : LINT := LINT#2147483647;
	MIN_VALUE_OF_LINT_WHICH_CAN_BE_HELD_IN_A_USINT : LINT := LINT#0;
	MAX_VALUE_OF_LINT_WHICH_CAN_BE_HELD_IN_A_USINT : LINT := LINT#255;
	MIN_VALUE_OF_LINT_WHICH_CAN_BE_HELD_IN_A_UINT : LINT := LINT#0;
	MAX_VALUE_OF_LINT_WHICH_CAN_BE_HELD_IN_A_UINT : LINT := LINT#65535;
	MIN_VALUE_OF_LINT_WHICH_CAN_BE_HELD_IN_A_UDINT : LINT := LINT#0;
	MAX_VALUE_OF_LINT_WHICH_CAN_BE_HELD_IN_A_UDINT : LINT := LINT#4294967295;
	MIN_VALUE_OF_LINT_WHICH_CAN_BE_HELD_IN_A_ULINT : LINT := LINT#0;
	MIN_VALUE_OF_LINT_WHICH_CAN_BE_HELD_IN_A_TIME : LINT := LINT#0;
	MAX_VALUE_OF_LINT_WHICH_CAN_BE_HELD_IN_A_TIME : LINT := LINT#4294967295;
	MIN_VALUE_OF_LINT_WHICH_CAN_BE_HELD_IN_A_TOD : LINT := LINT#0;
	MAX_VALUE_OF_LINT_WHICH_CAN_BE_HELD_IN_A_TOD : LINT := LINT#86399999;
	MIN_VALUE_OF_LINT_WHICH_CAN_BE_HELD_IN_A_DATE : LINT := LINT#0;
	MAX_VALUE_OF_LINT_WHICH_CAN_BE_HELD_IN_A_DATE : LINT := LINT#4294944000;
	MIN_VALUE_OF_LINT_WHICH_CAN_BE_HELD_IN_A_DT : LINT := LINT#0;
	MAX_VALUE_OF_LINT_WHICH_CAN_BE_HELD_IN_A_DT : LINT := LINT#4294967295;
	
	// Limits of USINT used for conversions
	MAX_VALUE_OF_USINT_WHICH_CAN_BE_HELD_IN_A_SINT : USINT := USINT#127;
	
	// Limits of UINT used for conversions
	MAX_VALUE_OF_UINT_WHICH_CAN_BE_HELD_IN_A_BYTE : UINT := UINT#255;
	MAX_VALUE_OF_UINT_WHICH_CAN_BE_HELD_IN_A_SINT : UINT := UINT#127;
	MAX_VALUE_OF_UINT_WHICH_CAN_BE_HELD_IN_A_INT : UINT := UINT#32767;
	MAX_VALUE_OF_UINT_WHICH_CAN_BE_HELD_IN_A_USINT : UINT := UINT#255;
	
	// Limits of UDINT used for conversions
	MAX_VALUE_OF_UDINT_WHICH_CAN_BE_HELD_IN_A_BYTE : UDINT := UDINT#255;
	MAX_VALUE_OF_UDINT_WHICH_CAN_BE_HELD_IN_A_WORD : UDINT := UDINT#65535;
	MAX_VALUE_OF_UDINT_WHICH_CAN_BE_HELD_IN_A_SINT : UDINT := UDINT#127;
	MAX_VALUE_OF_UDINT_WHICH_CAN_BE_HELD_IN_A_INT : UDINT := UDINT#32767;
	MAX_VALUE_OF_UDINT_WHICH_CAN_BE_HELD_IN_A_DINT : UDINT := UDINT#2147483647;
	MAX_VALUE_OF_UDINT_WHICH_CAN_BE_HELD_IN_A_USINT : UDINT := UDINT#255;
	MAX_VALUE_OF_UDINT_WHICH_CAN_BE_HELD_IN_A_UINT : UDINT := UDINT#65535;
	MAX_VALUE_OF_UDINT_WHICH_CAN_BE_HELD_IN_A_TOD : UDINT := UDINT#86399999;
	
	// Limits of ULINT used for conversions
	MAX_VALUE_OF_ULINT_WHICH_CAN_BE_HELD_IN_A_BYTE : ULINT := ULINT#255;
	MAX_VALUE_OF_ULINT_WHICH_CAN_BE_HELD_IN_A_WORD : ULINT := ULINT#65535;
	MAX_VALUE_OF_ULINT_WHICH_CAN_BE_HELD_IN_A_DWORD : ULINT := ULINT#4294967295;
	MAX_VALUE_OF_ULINT_WHICH_CAN_BE_HELD_IN_A_SINT : ULINT := ULINT#127;
	MAX_VALUE_OF_ULINT_WHICH_CAN_BE_HELD_IN_A_INT : ULINT := ULINT#32767;
	MAX_VALUE_OF_ULINT_WHICH_CAN_BE_HELD_IN_A_DINT : ULINT := ULINT#2147483647;
	MAX_VALUE_OF_ULINT_WHICH_CAN_BE_HELD_IN_A_LINT : ULINT := ULINT#9223372036854775807;
	MAX_VALUE_OF_ULINT_WHICH_CAN_BE_HELD_IN_A_USINT : ULINT := ULINT#255;
	MAX_VALUE_OF_ULINT_WHICH_CAN_BE_HELD_IN_A_UINT : ULINT := ULINT#65535;
	MAX_VALUE_OF_ULINT_WHICH_CAN_BE_HELD_IN_A_UDINT : ULINT := ULINT#4294967295;
	MAX_VALUE_OF_ULINT_WHICH_CAN_BE_HELD_IN_A_TIME : ULINT := ULINT#4294967295;
	MAX_VALUE_OF_ULINT_WHICH_CAN_BE_HELD_IN_A_TOD : ULINT := ULINT#86399999;
	MAX_VALUE_OF_ULINT_WHICH_CAN_BE_HELD_IN_A_DATE : ULINT := ULINT#4294944000;
	MAX_VALUE_OF_ULINT_WHICH_CAN_BE_HELD_IN_A_DT : ULINT := ULINT#4294967295;
	
	// Limits of REAL used for conversions
	MIN_VALUE_OF_REAL_WHICH_CAN_BE_HELD_IN_A_BYTE : REAL := REAL#0;
	MAX_VALUE_OF_REAL_WHICH_CAN_BE_HELD_IN_A_BYTE : REAL := REAL#255;
	MIN_VALUE_OF_REAL_WHICH_CAN_BE_HELD_IN_A_WORD : REAL := REAL#0;
	MAX_VALUE_OF_REAL_WHICH_CAN_BE_HELD_IN_A_WORD : REAL := REAL#65535;
	MIN_VALUE_OF_REAL_WHICH_CAN_BE_HELD_IN_A_DWORD : REAL := REAL#0;
	MAX_VALUE_OF_REAL_WHICH_CAN_BE_HELD_IN_A_DWORD : REAL := REAL#4.294967E+09;
	MIN_VALUE_OF_REAL_WHICH_CAN_BE_HELD_IN_A_LWORD : REAL := REAL#0;
	MAX_VALUE_OF_REAL_WHICH_CAN_BE_HELD_IN_A_LWORD : REAL := REAL#1.8446743E+19;
	MIN_VALUE_OF_REAL_WHICH_CAN_BE_HELD_IN_A_SINT : REAL := REAL#-128;
	MAX_VALUE_OF_REAL_WHICH_CAN_BE_HELD_IN_A_SINT : REAL := REAL#127;
	MIN_VALUE_OF_REAL_WHICH_CAN_BE_HELD_IN_A_INT : REAL := REAL#-32768;
	MAX_VALUE_OF_REAL_WHICH_CAN_BE_HELD_IN_A_INT : REAL := REAL#32767;
	MIN_VALUE_OF_REAL_WHICH_CAN_BE_HELD_IN_A_DINT : REAL := REAL#-2.14748352E+09;
	MAX_VALUE_OF_REAL_WHICH_CAN_BE_HELD_IN_A_DINT : REAL := REAL#2.14748352E+09;
	MIN_VALUE_OF_REAL_WHICH_CAN_BE_HELD_IN_A_LINT : REAL := REAL#-9.223372E+18;
	MAX_VALUE_OF_REAL_WHICH_CAN_BE_HELD_IN_A_LINT : REAL := REAL#9.223372E+18;
	MIN_VALUE_OF_REAL_WHICH_CAN_BE_HELD_IN_A_USINT : REAL := REAL#0;
	MAX_VALUE_OF_REAL_WHICH_CAN_BE_HELD_IN_A_USINT : REAL := REAL#255;
	MIN_VALUE_OF_REAL_WHICH_CAN_BE_HELD_IN_A_UINT : REAL := REAL#0;
	MAX_VALUE_OF_REAL_WHICH_CAN_BE_HELD_IN_A_UINT : REAL := REAL#65535;
	MIN_VALUE_OF_REAL_WHICH_CAN_BE_HELD_IN_A_UDINT : REAL := REAL#0;
	MAX_VALUE_OF_REAL_WHICH_CAN_BE_HELD_IN_A_UDINT : REAL := REAL#4.294967E+09;
	MIN_VALUE_OF_REAL_WHICH_CAN_BE_HELD_IN_A_ULINT : REAL := REAL#0;
	MAX_VALUE_OF_REAL_WHICH_CAN_BE_HELD_IN_A_ULINT : REAL := REAL#1.8446743E+19;
	MIN_VALUE_OF_REAL_WHICH_CAN_BE_HELD_IN_A_TIME : REAL := REAL#0;
	MAX_VALUE_OF_REAL_WHICH_CAN_BE_HELD_IN_A_TIME : REAL := REAL#4.294967E+09;
	MIN_VALUE_OF_REAL_WHICH_CAN_BE_HELD_IN_A_TOD : REAL := REAL#0;
	MAX_VALUE_OF_REAL_WHICH_CAN_BE_HELD_IN_A_TOD : REAL := REAL#8.639999E+07;
	MIN_VALUE_OF_REAL_WHICH_CAN_BE_HELD_IN_A_DATE : REAL := REAL#0;
	MAX_VALUE_OF_REAL_WHICH_CAN_BE_HELD_IN_A_DATE : REAL := REAL#4.294944E+09;
	MIN_VALUE_OF_REAL_WHICH_CAN_BE_HELD_IN_A_DT : REAL := REAL#0;
	MAX_VALUE_OF_REAL_WHICH_CAN_BE_HELD_IN_A_DT : REAL := REAL#4.294967E+09;
	
	// Limits of LREAL used for conversions
	MIN_VALUE_OF_LREAL_WHICH_CAN_BE_HELD_IN_A_BYTE : LREAL := LREAL#0;
	MAX_VALUE_OF_LREAL_WHICH_CAN_BE_HELD_IN_A_BYTE : LREAL := LREAL#255;
	MIN_VALUE_OF_LREAL_WHICH_CAN_BE_HELD_IN_A_WORD : LREAL := LREAL#0;
	MAX_VALUE_OF_LREAL_WHICH_CAN_BE_HELD_IN_A_WORD : LREAL := LREAL#65535;
	MIN_VALUE_OF_LREAL_WHICH_CAN_BE_HELD_IN_A_DWORD : LREAL := LREAL#0;
	MAX_VALUE_OF_LREAL_WHICH_CAN_BE_HELD_IN_A_DWORD : LREAL := LREAL#4294967295;
	MIN_VALUE_OF_LREAL_WHICH_CAN_BE_HELD_IN_A_LWORD : LREAL := LREAL#0;
	MAX_VALUE_OF_LREAL_WHICH_CAN_BE_HELD_IN_A_LWORD : LREAL := LREAL#1.844674407370955E+19;
	MIN_VALUE_OF_LREAL_WHICH_CAN_BE_HELD_IN_A_SINT : LREAL := LREAL#-128;
	MAX_VALUE_OF_LREAL_WHICH_CAN_BE_HELD_IN_A_SINT : LREAL := LREAL#127;
	MIN_VALUE_OF_LREAL_WHICH_CAN_BE_HELD_IN_A_INT : LREAL := LREAL#-32768;
	MAX_VALUE_OF_LREAL_WHICH_CAN_BE_HELD_IN_A_INT : LREAL := LREAL#32767;
	MIN_VALUE_OF_LREAL_WHICH_CAN_BE_HELD_IN_A_DINT : LREAL := LREAL#-2147483648;
	MAX_VALUE_OF_LREAL_WHICH_CAN_BE_HELD_IN_A_DINT : LREAL := LREAL#2147483647;
	MIN_VALUE_OF_LREAL_WHICH_CAN_BE_HELD_IN_A_LINT : LREAL := LREAL#-9.2233720368547758E+18;
	MAX_VALUE_OF_LREAL_WHICH_CAN_BE_HELD_IN_A_LINT : LREAL := LREAL#9.2233720368547758E+18;
	MIN_VALUE_OF_LREAL_WHICH_CAN_BE_HELD_IN_A_USINT : LREAL := LREAL#0;
	MAX_VALUE_OF_LREAL_WHICH_CAN_BE_HELD_IN_A_USINT : LREAL := LREAL#255;
	MIN_VALUE_OF_LREAL_WHICH_CAN_BE_HELD_IN_A_UINT : LREAL := LREAL#0;
	MAX_VALUE_OF_LREAL_WHICH_CAN_BE_HELD_IN_A_UINT : LREAL := LREAL#65535;
	MIN_VALUE_OF_LREAL_WHICH_CAN_BE_HELD_IN_A_UDINT : LREAL := LREAL#0;
	MAX_VALUE_OF_LREAL_WHICH_CAN_BE_HELD_IN_A_UDINT : LREAL := LREAL#4294967295;
	MIN_VALUE_OF_LREAL_WHICH_CAN_BE_HELD_IN_A_ULINT : LREAL := LREAL#0;
	MAX_VALUE_OF_LREAL_WHICH_CAN_BE_HELD_IN_A_ULINT : LREAL := LREAL#1.844674407370955E+19;
	MIN_VALUE_OF_LREAL_WHICH_CAN_BE_HELD_IN_A_REAL : LREAL := LREAL#-3.402823E+38;
	MAX_VALUE_OF_LREAL_WHICH_CAN_BE_HELD_IN_A_REAL : LREAL := LREAL#3.402823E+38;
	MIN_VALUE_OF_LREAL_WHICH_CAN_BE_HELD_IN_A_TIME : LREAL := LREAL#0;
	MAX_VALUE_OF_LREAL_WHICH_CAN_BE_HELD_IN_A_TIME : LREAL := LREAL#4294967295;
	MIN_VALUE_OF_LREAL_WHICH_CAN_BE_HELD_IN_A_TOD : LREAL := LREAL#0;
	MAX_VALUE_OF_LREAL_WHICH_CAN_BE_HELD_IN_A_TOD : LREAL := LREAL#86399999;
	MIN_VALUE_OF_LREAL_WHICH_CAN_BE_HELD_IN_A_DATE : LREAL := LREAL#0;
	MAX_VALUE_OF_LREAL_WHICH_CAN_BE_HELD_IN_A_DATE : LREAL := LREAL#4294944000;
	MIN_VALUE_OF_LREAL_WHICH_CAN_BE_HELD_IN_A_DT : LREAL := LREAL#0;
	MAX_VALUE_OF_LREAL_WHICH_CAN_BE_HELD_IN_A_DT : LREAL := LREAL#4294967295;
	MAX_VALUE_OF_LREAL_WHICH_CAN_BE_HELD_IN_A_STRING : LREAL := LREAL#9.999999999999E+307; // not sure why this is the number and not LREAL#4.94065645841247E-324.
	MIN_VALUE_OF_LREAL_WHICH_CAN_BE_HELD_IN_A_STRING : LREAL := LREAL#-9.999999999999E+307; // not sure why this is the number and not LREAL#-4.94065645841247E-324.
	
	// Limits of TIME used for conversions
	MAX_VALUE_OF_TIME_WHICH_CAN_BE_HELD_IN_A_BYTE : TIME := T#255MS;
	MAX_VALUE_OF_TIME_WHICH_CAN_BE_HELD_IN_A_WORD : TIME := T#1M5S535MS;
	MAX_VALUE_OF_TIME_WHICH_CAN_BE_HELD_IN_A_SINT : TIME := T#127MS;
	MAX_VALUE_OF_TIME_WHICH_CAN_BE_HELD_IN_A_INT : TIME := T#32S767MS;
	MAX_VALUE_OF_TIME_WHICH_CAN_BE_HELD_IN_A_DINT : TIME := T#24D20H31M23S647MS;
	MAX_VALUE_OF_TIME_WHICH_CAN_BE_HELD_IN_A_USINT : TIME := T#255MS;
	MAX_VALUE_OF_TIME_WHICH_CAN_BE_HELD_IN_A_UINT : TIME := T#1M5S535MS;
	MAX_VALUE_OF_TIME_WHICH_CAN_BE_HELD_IN_A_TOD : TIME := T#23H59M59S999MS;
	
	// Limits of TOD used for conversions
	MAX_VALUE_OF_TOD_WHICH_CAN_BE_HELD_IN_A_BYTE : TOD := TOD#0:0:0.255;
	MAX_VALUE_OF_TOD_WHICH_CAN_BE_HELD_IN_A_WORD : TOD := TOD#0:1:5.535;
	MAX_VALUE_OF_TOD_WHICH_CAN_BE_HELD_IN_A_SINT : TOD := TOD#0:0:0.127;
	MAX_VALUE_OF_TOD_WHICH_CAN_BE_HELD_IN_A_INT : TOD := TOD#0:0:32.767;
	MAX_VALUE_OF_TOD_WHICH_CAN_BE_HELD_IN_A_USINT : TOD := TOD#0:0:0.255;
	MAX_VALUE_OF_TOD_WHICH_CAN_BE_HELD_IN_A_UINT : TOD := TOD#0:1:5.535;
	
	// Limits of DATE used for conversions
	MAX_VALUE_OF_DATE_WHICH_CAN_BE_HELD_IN_A_BYTE : DATE := D#1970-1-1;
	MAX_VALUE_OF_DATE_WHICH_CAN_BE_HELD_IN_A_WORD : DATE := D#1970-1-1;
	MAX_VALUE_OF_DATE_WHICH_CAN_BE_HELD_IN_A_SINT : DATE := D#1970-1-1;
	MAX_VALUE_OF_DATE_WHICH_CAN_BE_HELD_IN_A_INT : DATE := D#1970-1-1;
	MAX_VALUE_OF_DATE_WHICH_CAN_BE_HELD_IN_A_DINT : DATE := D#2038-1-19;
	MAX_VALUE_OF_DATE_WHICH_CAN_BE_HELD_IN_A_USINT : DATE := D#1970-1-1;
	MAX_VALUE_OF_DATE_WHICH_CAN_BE_HELD_IN_A_UINT : DATE := D#1970-1-1;
	MAX_VALUE_OF_DATE_WHICH_CAN_BE_HELD_IN_A_TIME : DATE := D#1970-2-19;
	MAX_VALUE_OF_DATE_WHICH_CAN_BE_HELD_IN_A_TOD : DATE := D#1970-1-1;
	MAX_VALUE_OF_DATE_WHICH_CAN_BE_HELD_IN_A_DT : DATE := D#2106-2-7;
	
	// Limits of DT used for conversions
	MAX_VALUE_OF_DT_WHICH_CAN_BE_HELD_IN_A_BYTE : DT := DT#1970-1-1-0:4:15;
	MAX_VALUE_OF_DT_WHICH_CAN_BE_HELD_IN_A_WORD : DT := DT#1970-1-1-18:12:15;
	MAX_VALUE_OF_DT_WHICH_CAN_BE_HELD_IN_A_SINT : DT := DT#1970-1-1-0:2:7;
	MAX_VALUE_OF_DT_WHICH_CAN_BE_HELD_IN_A_INT : DT := DT#1970-1-1-9:6:7;
	MAX_VALUE_OF_DT_WHICH_CAN_BE_HELD_IN_A_DINT : DT := DT#2038-1-19-3:14:7;
	MAX_VALUE_OF_DT_WHICH_CAN_BE_HELD_IN_A_USINT : DT := DT#1970-1-1-0:4:15;
	MAX_VALUE_OF_DT_WHICH_CAN_BE_HELD_IN_A_UINT : DT := DT#1970-1-1-18:12:15;
	MAX_VALUE_OF_DT_WHICH_CAN_BE_HELD_IN_A_TIME : DT := DT#1970-2-19-17:2:47;
	MAX_VALUE_OF_DT_WHICH_CAN_BE_HELD_IN_A_TOD : DT := DT#1970-1-1-23:59:59;

END_VAR

// mobject-server/GVLs/ServerConfiguration
{attribute 'qualified_only'}
VAR_GLOBAL CONSTANT
	HEADER_STRING_SIZE : UDINT := 1024;
	PAYLOAD_STRING_SIZE : UDINT := 8000; // typically 1/8th of the Runtime Stack Size

	// Maximum time an asynchronous response may remain pending.
    // T#0S disables the deadline.
    PENDING_RESPONSE_MAX_AGE : TIME := T#60S;

    // Delay suggested to clients between asynchronous response polls.
    // Prevents clients continuously polling the PLC as fast as ADS allows.
    PENDING_RESPONSE_RETRY_DELAY_MS : UDINT := 20;
END_VAR

// mobject-collections/_Internal/Dictionary/Enumerator/DictionaryForwardEnumerator
{attribute 'linkalways'} 
{attribute 'no_explicit_call' := 'This FB is a CLASS and must be accessed using methods or properties'}
{attribute 'enable_dynamic_creation'}
FUNCTION_BLOCK DictionaryForwardEnumerator EXTENDS Disposable IMPLEMENTS I_KeyValueForwardEnumerator, I_EventHandler
VAR
	parent : I_Dictionary;
	nodes : I_Collection;
	collectionEnumerator : I_ForwardEnumerator;
	currentNode : I_DictionaryTreeNode;
	moveNextCalled : BOOL := FALSE;
	invalid : BOOL := FALSE; 
END_VAR

METHOD FB_init : BOOL
VAR_INPUT
	bInitRetains : BOOL; // if TRUE, the retain variables are initialized (warm start / cold start)
	bInCopyCode : BOOL;  // if TRUE, the instance afterwards gets moved into the copy code (online change)
	Parent : I_Dictionary;
	Nodes : I_Collection;
END_VAR
Parent.OnEvent('OnChanged',THIS^);
Parent.OnEvent('OnDisposed',THIS^);
THIS^.parent := Parent;
THIS^.nodes := Nodes;
THIS^.collectionEnumerator := Nodes.GetEnumerator();
END_METHOD

METHOD FB_exit : BOOL
VAR_INPUT
	bInCopyCode : BOOL; // if TRUE, the exit method is called for exiting an instance that is copied afterwards (online change).
END_VAR
IF bInCopyCode THEN
	RETURN;
END_IF

collectionEnumerator.Dispose();
nodes.Dispose();

IF parent = 0 THEN
	RETURN;
END_IF

parent.OffEvent('OnChanged',THIS^);
parent.OffEvent('OnDisposed',THIS^);
END_METHOD

METHOD PUBLIC HandleEvent
VAR_INPUT
	Event : I_Event;
END_VAR
VAR
	changedEvent : I_KeyValueCollectionChangedEvent;
	disposedEvent : I_KeyValueCollectionDisposedEvent;
END_VAR
IF __QUERYINTERFACE(Event, changedEvent) THEN
	invalid := TRUE;
	currentNode := 0;
ELSIF __QUERYINTERFACE(Event, disposedEvent) THEN
	parent := 0;	
	Dispose();
END_IF
END_METHOD

PROPERTY PUBLIC IsValid : BOOL
GET
PUBLIC
IsValid := (not invalid and parent <> 0);
END_GET
END_PROPERTY

PROPERTY PUBLIC Key : T_MAXSTRING
GET
IF NOT IsValid THEN
	RETURN;
END_IF

IF currentNode = 0 THEN
	RETURN;
END_IF

Key := currentNode.Key;
END_GET
END_PROPERTY

METHOD PUBLIC MoveNext : BOOL
IF invalid THEN
	RETURN;
END_IF

IF collectionEnumerator.MoveNext() THEN
	collectionEnumerator.TryGet(currentNode);
	MoveNext := TRUE;
END_IF
END_METHOD

METHOD Reset
VAR_INPUT
END_VAR
moveNextCalled := FALSE;
collectionEnumerator.Reset();
END_METHOD

METHOD PUBLIC TryGet : BOOL;
VAR_INPUT
	Destination : ANY;
END_VAR
IF currentNode <> 0 THEN
	TryGet := currentNode.TryGet(Destination);
END_IF
END_METHOD

METHOD PUBLIC TryGetTo : BOOL;
VAR_INPUT
	DestinationAddress : PVOID;
	DestinationSize : UDINT;
END_VAR
IF currentNode <> 0 THEN
	TryGetTo := currentNode.TryGetTo(DestinationAddress,DestinationSize);
END_IF
END_METHOD

END_FUNCTION_BLOCK

// mobject-disposable/Disposable/Disposable
{attribute 'linkalways'} 
{attribute 'no_explicit_call' := 'This FB is a CLASS and must be accessed using methods or properties'}
{attribute 'enable_dynamic_creation'}
FUNCTION_BLOCK ABSTRACT Disposable IMPLEMENTS I_Disposable
VAR
END_VAR

METHOD FB_exit : BOOL
VAR_INPUT
	bInCopyCode : BOOL; // if TRUE, the exit method is called for exiting an instance that is copied afterwards (online change).
END_VAR
// by default you would return if this is an in copy code, i.e. online change to this class
IF bInCopyCode THEN
	RETURN;
END_IF

// A word of warning. FB_exit does not NOT operate in the same way as a typical inherited method. If a child class does not implement FB_exit then it does not
// gain this one for itself. 
// The system will automatically call each FB_exit on each layer of inheritance one by one, starting with the child class and making it's way to the parent.
// Therefore code in here will only be triggered once the system reaches this layer of the object's deletion. The child class and all of it's variables
// will already have had FB_exit called by the time we reach this point!
END_METHOD

METHOD PUBLIC Dispose
VAR
	pDisposable : POINTER TO Disposable;
END_VAR
pDisposable := THIS;
__DELETE(pDisposable);
END_METHOD

END_FUNCTION_BLOCK

// mobject-disposable/Interfaces/I_Disposable
INTERFACE I_Disposable EXTENDS __System.IQueryInterface

METHOD PUBLIC Dispose
END_METHOD

END_INTERFACE

// mobject-enumerable/Interfaces/Enumerators/I_KeyValueForwardEnumerator
INTERFACE I_KeyValueForwardEnumerator EXTENDS I_ForwardEnumerator

PROPERTY Key : T_MAXSTRING
GET
END_GET
END_PROPERTY

END_INTERFACE

// mobject-enumerable/Interfaces/Enumerators/I_ForwardEnumerator
INTERFACE I_ForwardEnumerator EXTENDS I_Disposable

PROPERTY PUBLIC IsValid : BOOL
GET
END_GET
END_PROPERTY

METHOD PUBLIC MoveNext : BOOL
END_METHOD

METHOD PUBLIC Reset
END_METHOD

METHOD PUBLIC TryGet : BOOL;
VAR_INPUT
    Destination : ANY;
END_VAR
END_METHOD

METHOD PUBLIC TryGetTo : BOOL;
VAR_INPUT
    DestinationAddress : PVOID;
    DestinationSize : UDINT;
END_VAR
END_METHOD

END_INTERFACE

// mobject-events/Interfaces/I_EventHandler
INTERFACE I_EventHandler EXTENDS __SYSTEM.IQueryInterface

METHOD PUBLIC HandleEvent
VAR_INPUT
	Event : I_Event;
END_VAR
END_METHOD

END_INTERFACE

// mobject-events/Interfaces/I_Event
INTERFACE I_Event EXTENDS __SYSTEM.IQueryInterface

END_INTERFACE

// mobject-collections/Interfaces/KeyValueCollections/I_Dictionary
INTERFACE I_Dictionary EXTENDS I_KeyValueCollection

METHOD PUBLIC AddOrUpdate
VAR_INPUT
	Key : T_MAXSTRING;
	Value : ANY;
END_VAR
END_METHOD

METHOD PUBLIC Clear
VAR_INPUT
END_VAR
END_METHOD

METHOD PUBLIC ContainsKey : BOOL
VAR_INPUT
	Key : T_MAXSTRING;
END_VAR
END_METHOD

METHOD PUBLIC GetKeys : I_Collection
END_METHOD

PROPERTY IsEmpty : BOOL
GET
END_GET
END_PROPERTY

METHOD PUBLIC Remove
VAR_INPUT
	Key : T_MAXSTRING;
END_VAR
END_METHOD

METHOD PUBLIC TryAdd : BOOL
VAR_INPUT
	Key : T_MAXSTRING;
	Value : ANY;
END_VAR
END_METHOD

METHOD PUBLIC TryGetValue : BOOL
VAR_INPUT
	Key : T_MAXSTRING;
	Destination	: ANY;
END_VAR
END_METHOD

METHOD PUBLIC TryGetValueTo : BOOL
VAR_INPUT
	Key : T_MAXSTRING;
	DestinationAddress : PVOID;
	DestinationSize : UDINT;
END_VAR
END_METHOD

END_INTERFACE

// mobject-collections/Interfaces/KeyValueCollections/I_KeyValueCollection
INTERFACE I_KeyValueCollection EXTENDS I_KeyValueEnumerable, I_Enumerable, I_Disposable, I_EventEmitter

END_INTERFACE

// mobject-enumerable/Interfaces/I_KeyValueEnumerable
INTERFACE I_KeyValueEnumerable EXTENDS __SYSTEM.IQueryInterface

METHOD PUBLIC GetKeyValueEnumerator : I_KeyValueForwardEnumerator
END_METHOD

END_INTERFACE

// mobject-enumerable/Interfaces/I_Enumerable
INTERFACE I_Enumerable EXTENDS __SYSTEM.IQueryInterface

METHOD PUBLIC GetEnumerator : I_ForwardEnumerator
END_METHOD

END_INTERFACE

// mobject-events/Interfaces/I_EventEmitter
INTERFACE I_EventEmitter EXTENDS __SYSTEM.IQueryInterface

METHOD PUBLIC OffEvent
VAR_INPUT
	EventName : T_MaxString;
	EventHandler : I_EventHandler;
END_VAR
END_METHOD

METHOD PUBLIC OnceEvent
VAR_INPUT
	EventName : T_MaxString;
	EventHandler : I_EventHandler;
END_VAR
END_METHOD

METHOD PUBLIC OnEvent
VAR_INPUT
	EventName : T_MaxString;
	EventHandler : I_EventHandler;
END_VAR
END_METHOD

END_INTERFACE

// mobject-collections/Interfaces/Collections/I_Collection
INTERFACE I_Collection EXTENDS I_Enumerable, I_Disposable, I_EventEmitter

METHOD PUBLIC AddItem
VAR_INPUT
	Item : ANY;
END_VAR
END_METHOD

METHOD PUBLIC Clear
END_METHOD

METHOD PUBLIC Contains : BOOL;
VAR_INPUT
	Item : ANY;
END_VAR
END_METHOD

PROPERTY PUBLIC Count : DINT
GET
END_GET
END_PROPERTY

PROPERTY IsEmpty : BOOL
GET
END_GET
END_PROPERTY

METHOD PUBLIC TryCopyTo : BOOL
VAR_INPUT
	Destination : ANY;
END_VAR
END_METHOD

METHOD PUBLIC TryCopyToLocation : BOOL
VAR_INPUT
	DestinationAddress : PVOID;
	DestinationSize : UDINT;
END_VAR
END_METHOD

METHOD PUBLIC TryRemoveItem : BOOL
VAR_INPUT
	Item : ANY;
END_VAR
END_METHOD

END_INTERFACE

// mobject-collections/Interfaces/KeyValueCollections/Nodes/I_DictionaryTreeNode
INTERFACE I_DictionaryTreeNode EXTENDS I_CollectionNode

METHOD PUBLIC DeepCopy
VAR_INPUT
	Node : I_DictionaryTreeNode;
END_VAR
END_METHOD

PROPERTY PUBLIC Height : DINT
GET
END_GET
SET
END_SET
END_PROPERTY

PROPERTY PUBLIC Key : T_MAXSTRING
GET
END_GET
END_PROPERTY

PROPERTY PUBLIC Left : I_DictionaryTreeNode
GET
END_GET
SET
END_SET
END_PROPERTY

PROPERTY PUBLIC NodeBufferPointer : Pointer To Byte
GET
END_GET
END_PROPERTY

PROPERTY PUBLIC NodeBufferSize : UDINT
GET
END_GET
END_PROPERTY

METHOD Reinitialize
VAR_INPUT
	Key : T_MAXSTRING;
	Source : ANY;
END_VAR
END_METHOD

PROPERTY PUBLIC Right : I_DictionaryTreeNode
GET
END_GET
SET
END_SET
END_PROPERTY

END_INTERFACE

// mobject-collections/Interfaces/Collections/Nodes/I_CollectionNode
INTERFACE I_CollectionNode EXTENDS I_Disposable

PROPERTY PUBLIC DataSize : UDINT
GET
END_GET
END_PROPERTY

METHOD PUBLIC Equals : BOOL
VAR_INPUT
	Symbol : ANY;
END_VAR
END_METHOD

METHOD PUBLIC TryGet : BOOL;
VAR_INPUT
	Destination : ANY;
END_VAR
END_METHOD

METHOD PUBLIC TryGetTo : BOOL;
VAR_INPUT
	DestinationAddress : PVOID;
	DestinationSize : UDINT;
END_VAR
END_METHOD

END_INTERFACE

// mobject-collections/Interfaces/KeyValueCollections/Events/I_KeyValueCollectionChangedEvent
INTERFACE I_KeyValueCollectionChangedEvent EXTENDS I_Event

PROPERTY PUBLIC Target : I_KeyValueCollection
GET
END_GET
END_PROPERTY

END_INTERFACE

// mobject-collections/Interfaces/KeyValueCollections/Events/I_KeyValueCollectionDisposedEvent
INTERFACE I_KeyValueCollectionDisposedEvent EXTENDS I_Event

PROPERTY PUBLIC Target : I_KeyValueCollection
GET
END_GET
END_PROPERTY

END_INTERFACE

// mobject-collections/_Internal/Dictionary/Node/DictionaryTreeNode
{attribute 'linkalways'} 
{attribute 'no_explicit_call' := 'This FB is a CLASS and must be accessed using methods or properties'}
{attribute 'enable_dynamic_creation'}
FUNCTION_BLOCK DictionaryTreeNode EXTENDS Disposable IMPLEMENTS I_DictionaryTreeNode
VAR
	_key : T_MAXSTRING;
	pBuffer : POINTER TO BYTE;
	bufferSize : UDINT;
    _height : DINT;
    _left : I_DictionaryTreeNode;
    _right : I_DictionaryTreeNode;
END_VAR

METHOD FB_init : BOOL
VAR_INPUT
	bInitRetains : BOOL; // if TRUE, the retain variables are initialized (warm start / cold start)
	bInCopyCode : BOOL;  // if TRUE, the instance afterwards gets moved into the copy code (online change)
	NodeKey : T_MAXSTRING;
	NodeSource : ANY;
END_VAR
_key := NodeKey;
CreateBuffer(DINT_TO_UDINT(NodeSource.diSize));
CopySourceToBuffer(NodeSource.pValue);
END_METHOD

METHOD FB_exit : BOOL
VAR_INPUT
	bInCopyCode : BOOL; // if TRUE, the exit method is called for exiting an instance that is copied afterwards (online change).
END_VAR
IF bInCopyCode THEN
	RETURN;
END_IF

DestroyBuffer();
END_METHOD

METHOD PRIVATE CopyBufferToDestination
VAR_INPUT
	DestinationAddress : PVOID;
END_VAR
MEMCPY(DestinationAddress, pBuffer, bufferSize);
END_METHOD

METHOD PRIVATE CopySourceToBuffer
VAR_INPUT
	SourceAddress : PVOID;
END_VAR
MEMCPY(pBuffer, SourceAddress, bufferSize);
END_METHOD

METHOD PRIVATE CreateBuffer
VAR_INPUT
	SizeInBytes : UDINT;
END_VAR
bufferSize := SizeInBytes;
pBuffer := __NEW(BYTE, SizeInBytes);
END_METHOD

METHOD PRIVATE DestroyBuffer
VAR_INPUT
END_VAR
IF pBuffer = 0 THEN
	RETURN;
END_IF

__DELETE(pBuffer);
bufferSize := 0;
END_METHOD

PROPERTY PUBLIC DataSize : UDINT
GET
DataSize := bufferSize;
END_GET
END_PROPERTY

METHOD PUBLIC DeepCopy
VAR_INPUT
	Node : I_DictionaryTreeNode;
END_VAR
DestroyBuffer();
CreateBuffer(Node.NodeBufferSize);
CopySourceToBuffer(Node.NodeBufferPointer);
_key := Node.Key;
END_METHOD

METHOD PUBLIC Equals : BOOL
VAR_INPUT
	Symbol : ANY;
END_VAR
IF pBuffer = 0 THEN
	RETURN;
END_IF

IF bufferSize <> DINT_TO_UDINT(symbol.diSize) THEN
	RETURN;
END_IF

Equals := MEMCMP(Symbol.pValue, pBuffer, bufferSize) = 0;
END_METHOD

PROPERTY PUBLIC Height : DINT
GET
Height := _height;
END_GET
SET
PUBLIC 
VAR
END_VAR
_height := Height;
END_SET
END_PROPERTY

PROPERTY PUBLIC Key : T_MAXSTRING
GET
Key := _key;
END_GET
END_PROPERTY

PROPERTY PUBLIC Left : I_DictionaryTreeNode
GET
Left := _left;
END_GET
SET
_left := Left;
END_SET
END_PROPERTY

PROPERTY PUBLIC NodeBufferPointer : Pointer To Byte
GET
NodeBufferPointer := pBuffer;
END_GET
END_PROPERTY

PROPERTY PUBLIC NodeBufferSize : UDINT
GET
NodeBufferSize := bufferSize;
END_GET
END_PROPERTY

METHOD Reinitialize
VAR_INPUT
	Key : T_MAXSTRING;
	Source : ANY;
END_VAR
_key := Key;

IF pBuffer <> 0 THEN
	DestroyBuffer();
END_IF

CreateBuffer(DINT_TO_UDINT(Source.diSize));
CopySourceToBuffer(Source.pValue);
END_METHOD

PROPERTY PUBLIC Right : I_DictionaryTreeNode
GET
Right := _right;
END_GET
SET
_right := Right;
END_SET
END_PROPERTY

METHOD TryGet : BOOL
VAR_INPUT
	Destination	: ANY;
END_VAR
TryGet := TryGetTo(Destination.pValue, DINT_TO_UDINT(Destination.diSize));
END_METHOD

METHOD TryGetTo : BOOL
VAR_INPUT
	DestinationAddress : PVOID;
	DestinationSize : UDINT;
END_VAR
IF pBuffer = 0 THEN
	RETURN;
END_IF

IF bufferSize <> DestinationSize THEN
	RETURN;
END_IF

CopyBufferToDestination(DestinationAddress);
TryGetTo := TRUE;
END_METHOD

END_FUNCTION_BLOCK

// mobject-collections/_Internal/Events/Collection/CollectionChangedEvent
{attribute 'linkalways'} 
{attribute 'no_explicit_call' := 'This FB is a CLASS and must be accessed using methods or properties'}
{attribute 'enable_dynamic_creation'}
FUNCTION_BLOCK CollectionChangedEvent EXTENDS CollectionEvent IMPLEMENTS I_CollectionChangedEvent

END_FUNCTION_BLOCK

